LIN {X 0,Y 509.342,Z 622.742,A -85,B 0,C 180,E1 -5495.94,E2 -5495.94} C_VEL
LIN {X 0,Y 509.421,Z 617.168,A -85,B 0,C 180,E1 -5497.133,E2 -5497.133} C_VEL
LIN {X 0,Y 509.56,Z 611.515,A -85,B 0,C 180,E1 -5498.127,E2 -5498.127} C_VEL
LIN {X 0,Y 509.746,Z 604.71,A -85,B 0,C 180,E1 -5499.123,E2 -5499.123} C_VEL
LIN {X 0,Y 509.975,Z 596.49,A -85,B 0,C 180,E1 -5500.12,E2 -5500.12} C_VEL
LIN {X 0,Y 510.261,Z 588.661,A -85,B 0,C 180,E1 -5500.917,E2 -5500.917} C_VEL
LIN {X 0,Y 510.548,Z 580.574,A -85,B 0,C 180,E1 -5501.614,E2 -5501.614} C_VEL
LIN {X 0,Y 510.783,Z 570.465,A -85,B 0,C 180,E1 -5502.336,E2 -5502.336} C_VEL
LIN {X 0,Y 511.032,Z 562.413,A -85,B 0,C 180,E1 -5502.813,E2 -5502.813} C_VEL
LIN {X 0,Y 511.32,Z 551.902,A -85,B 0,C 180,E1 -5503.31,E2 -5503.31} C_VEL
LIN {X 0,Y 511.513,Z 541.564,A -85,B 0,C 180,E1 -5503.685,E2 -5503.685} C_VEL
LIN {X 0,Y 511.738,Z 530.84,A -85,B 0,C 180,E1 -5503.957,E2 -5503.957} C_VEL
LIN {X 0,Y 511.952,Z 508.063,A -85,B 0,C 180,E1 -5504.306,E2 -5504.306} C_VEL
LIN {X 0,Y 512.118,Z 435.713,A -85,B 0,C 180,E1 -5505.329,E2 -5505.329} C_VEL
LIN {X 0,Y 510.056,Z 423.426,A -85,B 0,C 180,E1 -5505.593,E2 -5505.593} C_VEL
LIN {X 0,Y 510.461,Z 407.833,A -85,B 0,C 180,E1 -5508.669,E2 -5508.669} C_VEL
LIN {X 0,Y 510.875,Z 391.094,A -85,B 0,C 180,E1 -5512.016,E2 -5512.016} C_VEL
LIN {X 0,Y 511.227,Z 378.573,A -85,B 0,C 180,E1 -5514.597,E2 -5514.597} C_VEL
LIN {X 0,Y 509.916,Z 370.577,A -85,B 0,C 180,E1 -5516.406,E2 -5516.406} C_VEL
LIN {X 0,Y 509.885,Z 370.471,A -85,B 0,C 180,E1 -5518.844,E2 -5518.844} C_VEL
LIN {X 0,Y 509.826,Z 370.48,A -85,B 0,C 180,E1 -5521.59,E2 -5521.59} C_VEL
LIN {X 0,Y 509.857,Z 370.474,A -85,B 0,C 180,E1 -5524.413,E2 -5524.413} C_VEL
LIN {X 0,Y 509.822,Z 370.475,A -85,B 0,C 180,E1 -5527.34,E2 -5527.34} C_VEL
LIN {X 0,Y 509.84,Z 370.468,A -85,B 0,C 180,E1 -5530.382,E2 -5530.382} C_VEL
LIN {X 0,Y 509.825,Z 370.474,A -85,B 0,C 180,E1 -5533.062,E2 -5533.062} C_VEL
LIN {X 0,Y 509.832,Z 370.478,A -85,B 0,C 180,E1 -5535.792,E2 -5535.792} C_VEL
LIN {X 0,Y 509.867,Z 370.469,A -85,B 0,C 180,E1 -5538.575,E2 -5538.575} C_VEL
LIN {X 0,Y 509.853,Z 370.475,A -85,B 0,C 180,E1 -5541.786,E2 -5541.786} C_VEL
LIN {X 0,Y 509.843,Z 370.47,A -85,B 0,C 180,E1 -5544.622,E2 -5544.622} C_VEL
LIN {X 0,Y 509.866,Z 370.468,A -85,B 0,C 180,E1 -5547.481,E2 -5547.481} C_VEL
LIN {X 0,Y 509.882,Z 370.469,A -85,B 0,C 180,E1 -5550.268,E2 -5550.268} C_VEL
LIN {X 0,Y 509.885,Z 370.459,A -85,B 0,C 180,E1 -5552.944,E2 -5552.944} C_VEL
LIN {X 0,Y 509.869,Z 370.47,A -85,B 0,C 180,E1 -5555.574,E2 -5555.574} C_VEL
LIN {X 0,Y 509.821,Z 370.477,A -85,B 0,C 180,E1 -5558.148,E2 -5558.148} C_VEL
LIN {X 0,Y 509.864,Z 370.461,A -85,B 0,C 180,E1 -5560.681,E2 -5560.681} C_VEL
LIN {X 0,Y 509.884,Z 370.462,A -85,B 0,C 180,E1 -5563.174,E2 -5563.174} C_VEL
LIN {X 0,Y 509.863,Z 370.475,A -85,B 0,C 180,E1 -5565.634,E2 -5565.634} C_VEL
LIN {X 0,Y 509.911,Z 370.458,A -85,B 0,C 180,E1 -5568.874,E2 -5568.874} C_VEL
LIN {X 0,Y 509.95,Z 370.458,A -85,B 0,C 180,E1 -5572.078,E2 -5572.078} C_VEL
LIN {X 0,Y 509.98,Z 370.455,A -85,B 0,C 180,E1 -5574.464,E2 -5574.464} C_VEL
LIN {X 0,Y 510.053,Z 370.45,A -85,B 0,C 180,E1 -5577.63,E2 -5577.63} C_VEL
LIN {X 0,Y 510.062,Z 370.433,A -85,B 0,C 180,E1 -5580.789,E2 -5580.789} C_VEL
LIN {X 0,Y 509.955,Z 370.457,A -85,B 0,C 180,E1 -5583.16,E2 -5583.16} C_VEL
LIN {X 0,Y 509.975,Z 370.455,A -85,B 0,C 180,E1 -5586.329,E2 -5586.329} C_VEL
LIN {X 0,Y 509.913,Z 370.457,A -85,B 0,C 180,E1 -5588.72,E2 -5588.72} C_VEL
LIN {X 0,Y 509.948,Z 370.46,A -85,B 0,C 180,E1 -5591.93,E2 -5591.93} C_VEL
LIN {X 0,Y 509.89,Z 370.471,A -85,B 0,C 180,E1 -5595.241,E2 -5595.241} C_VEL
LIN {X 0,Y 509.885,Z 370.461,A -85,B 0,C 180,E1 -5598.001,E2 -5598.001} C_VEL
LIN {X 0,Y 509.847,Z 370.468,A -85,B 0,C 180,E1 -5601.001,E2 -5601.001} C_VEL
LIN {X 0,Y 509.866,Z 370.469,A -85,B 0,C 180,E1 -5604.426,E2 -5604.426} C_VEL
LIN {X 0,Y 509.884,Z 370.465,A -85,B 0,C 180,E1 -5607.055,E2 -5607.055} C_VEL
LIN {X 0,Y 509.853,Z 370.475,A -85,B 0,C 180,E1 -5609.751,E2 -5609.751} C_VEL
LIN {X 0,Y 509.873,Z 370.469,A -85,B 0,C 180,E1 -5612.775,E2 -5612.775} C_VEL
LIN {X 0,Y 509.838,Z 370.478,A -85,B 0,C 180,E1 -5615.581,E2 -5615.581} C_VEL
LIN {X 0,Y 509.846,Z 370.472,A -85,B 0,C 180,E1 -5618.338,E2 -5618.338} C_VEL
LIN {X 0,Y 509.855,Z 370.475,A -85,B 0,C 180,E1 -5621.425,E2 -5621.425} C_VEL
LIN {X 0,Y 509.852,Z 370.471,A -85,B 0,C 180,E1 -5624.668,E2 -5624.668} C_VEL
LIN {X 0,Y 509.857,Z 370.456,A -85,B 0,C 180,E1 -5628.102,E2 -5628.102} C_VEL
LIN {X 0,Y 509.856,Z 370.469,A -85,B 0,C 180,E1 -5630.649,E2 -5630.649} C_VEL
LIN {X 0,Y 509.828,Z 370.472,A -85,B 0,C 180,E1 -5633.742,E2 -5633.742} C_VEL
LIN {X 0,Y 509.162,Z 370.553,A -85,B 0,C 180,E1 -5634.402,E2 -5634.402} C_VEL
LIN {X 0,Y 506.344,Z 370.904,A -85,B 0,C 180,E1 -5635.474,E2 -5635.474} C_VEL
LIN {X 0,Y 503.951,Z 371.205,A -85,B 0,C 180,E1 -5636.337,E2 -5636.337} C_VEL
LIN {X 0,Y 502.902,Z 371.337,A -85,B 0,C 180,E1 -5637.004,E2 -5637.004} C_VEL
LIN {X 0,Y 502.805,Z 371.348,A -85,B 0,C 180,E1 -5637.229,E2 -5637.229} C_VEL
LIN {X 0,Y 502.827,Z 371.341,A -85,B 0,C 180,E1 -5640.061,E2 -5640.061} C_VEL
LIN {X 0,Y 502.831,Z 371.347,A -85,B 0,C 180,E1 -5642.533,E2 -5642.533} C_VEL
LIN {X 0,Y 502.825,Z 371.354,A -85,B 0,C 180,E1 -5645.298,E2 -5645.298} C_VEL
LIN {X 0,Y 502.79,Z 371.354,A -85,B 0,C 180,E1 -5647.827,E2 -5647.827} C_VEL
LIN {X 0,Y 502.823,Z 371.349,A -85,B 0,C 180,E1 -5650.4,E2 -5650.4} C_VEL
LIN {X 0,Y 502.831,Z 371.353,A -85,B 0,C 180,E1 -5652.932,E2 -5652.932} C_VEL
LIN {X 0,Y 502.842,Z 371.351,A -85,B 0,C 180,E1 -5655.429,E2 -5655.429} C_VEL
LIN {X 0,Y 502.874,Z 371.347,A -85,B 0,C 180,E1 -5658.717,E2 -5658.717} C_VEL
LIN {X 0,Y 502.898,Z 371.34,A -85,B 0,C 180,E1 -5661.966,E2 -5661.966} C_VEL
LIN {X 0,Y 502.939,Z 371.336,A -85,B 0,C 180,E1 -5664.386,E2 -5664.386} C_VEL
LIN {X 0,Y 503.023,Z 371.326,A -85,B 0,C 180,E1 -5667.598,E2 -5667.598} C_VEL
LIN {X 0,Y 503.025,Z 371.324,A -85,B 0,C 180,E1 -5670,E2 -5670} C_VEL
LIN {X 0,Y 503.022,Z 371.326,A -85,B 0,C 180,E1 -5672.402,E2 -5672.402} C_VEL
LIN {X 0,Y 502.939,Z 371.336,A -85,B 0,C 180,E1 -5675.613,E2 -5675.613} C_VEL
LIN {X 0,Y 502.898,Z 371.34,A -85,B 0,C 180,E1 -5678.033,E2 -5678.033} C_VEL
LIN {X 0,Y 502.873,Z 371.347,A -85,B 0,C 180,E1 -5681.283,E2 -5681.283} C_VEL
LIN {X 0,Y 502.841,Z 371.351,A -85,B 0,C 180,E1 -5684.571,E2 -5684.571} C_VEL
LIN {X 0,Y 502.858,Z 371.344,A -85,B 0,C 180,E1 -5687.907,E2 -5687.907} C_VEL
LIN {X 0,Y 502.824,Z 371.353,A -85,B 0,C 180,E1 -5690.536,E2 -5690.536} C_VEL
LIN {X 0,Y 502.792,Z 371.358,A -85,B 0,C 180,E1 -5693.04,E2 -5693.04} C_VEL
LIN {X 0,Y 502.837,Z 371.347,A -85,B 0,C 180,E1 -5695.675,E2 -5695.675} C_VEL
LIN {X 0,Y 502.837,Z 371.349,A -85,B 0,C 180,E1 -5698.372,E2 -5698.372} C_VEL
LIN {X 0,Y 502.791,Z 371.352,A -85,B 0,C 180,E1 -5701.499,E2 -5701.499} C_VEL
LIN {X 0,Y 502.8,Z 371.346,A -85,B 0,C 180,E1 -5704.444,E2 -5704.444} C_VEL
LIN {X 0,Y 502.775,Z 371.356,A -85,B 0,C 180,E1 -5707.178,E2 -5707.178} C_VEL
LIN {X 0,Y 502.815,Z 371.346,A -85,B 0,C 180,E1 -5710.012,E2 -5710.012} C_VEL
LIN {X 0,Y 502.766,Z 371.348,A -85,B 0,C 180,E1 -5713.231,E2 -5713.231} C_VEL
LIN {X 0,Y 502.783,Z 371.351,A -85,B 0,C 180,E1 -5715.661,E2 -5715.661} C_VEL
LIN {X 0,Y 502.813,Z 371.348,A -85,B 0,C 180,E1 -5718.934,E2 -5718.934} C_VEL
LIN {X 0,Y 502.788,Z 371.353,A -85,B 0,C 180,E1 -5722.046,E2 -5722.046} C_VEL
LIN {X 0,Y 502.803,Z 371.345,A -85,B 0,C 180,E1 -5725.035,E2 -5725.035} C_VEL
LIN {X 0,Y 502.781,Z 371.352,A -85,B 0,C 180,E1 -5727.916,E2 -5727.916} C_VEL
LIN {X 0,Y 502.832,Z 371.347,A -85,B 0,C 180,E1 -5730.713,E2 -5730.713} C_VEL
LIN {X 0,Y 502.874,Z 371.335,A -85,B 0,C 180,E1 -5733.435,E2 -5733.435} C_VEL
LIN {X 0,Y 502.784,Z 371.354,A -85,B 0,C 180,E1 -5736.086,E2 -5736.086} C_VEL
LIN {X 0,Y 502.777,Z 371.353,A -85,B 0,C 180,E1 -5738.689,E2 -5738.689} C_VEL
LIN {X 0,Y 502.824,Z 371.338,A -85,B 0,C 180,E1 -5741.249,E2 -5741.249} C_VEL
LIN {X 0,Y 502.817,Z 371.346,A -85,B 0,C 180,E1 -5743.767,E2 -5743.767} C_VEL
LIN {X 0,Y 502.825,Z 371.352,A -85,B 0,C 180,E1 -5746.255,E2 -5746.255} C_VEL
LIN {X 0,Y 502.886,Z 371.333,A -85,B 0,C 180,E1 -5748.718,E2 -5748.718} C_VEL
LIN {X 0,Y 502.895,Z 371.334,A -85,B 0,C 180,E1 -5751.967,E2 -5751.967} C_VEL
LIN {X 0,Y 502.933,Z 371.341,A -85,B 0,C 180,E1 -5754.387,E2 -5754.387} C_VEL
LIN {X 0,Y 503.02,Z 371.318,A -85,B 0,C 180,E1 -5757.598,E2 -5757.598} C_VEL
LIN {X 0,Y 503.021,Z 371.313,A -85,B 0,C 180,E1 -5760,E2 -5760} C_VEL
LIN {X 0,Y 503.02,Z 371.327,A -85,B 0,C 180,E1 -5762.403,E2 -5762.403} C_VEL
LIN {X 0,Y 502.934,Z 371.333,A -85,B 0,C 180,E1 -5765.614,E2 -5765.614} C_VEL
LIN {X 0,Y 502.896,Z 371.338,A -85,B 0,C 180,E1 -5768.034,E2 -5768.034} C_VEL
LIN {X 0,Y 502.872,Z 371.335,A -85,B 0,C 180,E1 -5771.284,E2 -5771.284} C_VEL
LIN {X 0,Y 502.84,Z 371.347,A -85,B 0,C 180,E1 -5774.571,E2 -5774.571} C_VEL
LIN {X 0,Y 502.857,Z 371.339,A -85,B 0,C 180,E1 -5777.908,E2 -5777.908} C_VEL
LIN {X 0,Y 502.824,Z 371.348,A -85,B 0,C 180,E1 -5780.537,E2 -5780.537} C_VEL
LIN {X 0,Y 502.792,Z 371.35,A -85,B 0,C 180,E1 -5783.041,E2 -5783.041} C_VEL
LIN {X 0,Y 502.838,Z 371.343,A -85,B 0,C 180,E1 -5785.676,E2 -5785.676} C_VEL
LIN {X 0,Y 502.839,Z 371.349,A -85,B 0,C 180,E1 -5788.373,E2 -5788.373} C_VEL
LIN {X 0,Y 502.794,Z 371.351,A -85,B 0,C 180,E1 -5791.5,E2 -5791.5} C_VEL
LIN {X 0,Y 502.804,Z 371.35,A -85,B 0,C 180,E1 -5794.446,E2 -5794.446} C_VEL
LIN {X 0,Y 502.779,Z 371.352,A -85,B 0,C 180,E1 -5797.179,E2 -5797.179} C_VEL
LIN {X 0,Y 502.82,Z 371.35,A -85,B 0,C 180,E1 -5800.013,E2 -5800.013} C_VEL
LIN {X 0,Y 502.821,Z 371.353,A -85,B 0,C 180,E1 -5802.203,E2 -5802.203} C_VEL
LIN {X 0,Y 502.799,Z 371.351,A -85,B 0,C 180,E1 -5805.469,E2 -5805.469} C_VEL
LIN {X 0,Y 502.82,Z 371.339,A -85,B 0,C 180,E1 -5808.935,E2 -5808.935} C_VEL
LIN {X 0,Y 502.794,Z 371.358,A -85,B 0,C 180,E1 -5812.047,E2 -5812.047} C_VEL
LIN {X 0,Y 502.81,Z 371.348,A -85,B 0,C 180,E1 -5815.036,E2 -5815.036} C_VEL
LIN {X 0,Y 502.786,Z 371.356,A -85,B 0,C 180,E1 -5817.916,E2 -5817.916} C_VEL
LIN {X 0,Y 502.841,Z 371.349,A -85,B 0,C 180,E1 -5820.714,E2 -5820.714} C_VEL
LIN {X 0,Y 502.867,Z 371.475,A -85,B 0,C 180,E1 -5823.439,E2 -5823.439} C_VEL
LIN {X 0,Y 504.25,Z 379.576,A -85,B 0,C 180,E1 -5825.284,E2 -5825.284} C_VEL
LIN {X 0,Y 503.892,Z 393.054,A -85,B 0,C 180,E1 -5828.094,E2 -5828.094} C_VEL
LIN {X 0,Y 503.435,Z 408.697,A -85,B 0,C 180,E1 -5831.272,E2 -5831.272} C_VEL
LIN {X 0,Y 503.026,Z 423.045,A -85,B 0,C 180,E1 -5834.167,E2 -5834.167} C_VEL
LIN {X 0,Y 503.739,Z 427.556,A -85,B 0,C 180,E1 -5834.295,E2 -5834.295} C_VEL
LIN {X 0,Y 505.36,Z 437.202,A -85,B 0,C 180,E1 -5834.486,E2 -5834.486} C_VEL
LIN {X 0,Y 504.882,Z 528.027,A -85,B 0,C 180,E1 -5835.798,E2 -5835.798} C_VEL
LIN {X 0,Y 504.693,Z 537.941,A -85,B 0,C 180,E1 -5836.024,E2 -5836.024} C_VEL
LIN {X 0,Y 504.506,Z 547.93,A -85,B 0,C 180,E1 -5836.353,E2 -5836.353} C_VEL
LIN {X 0,Y 504.175,Z 558.287,A -85,B 0,C 180,E1 -5836.806,E2 -5836.806} C_VEL
LIN {X 0,Y 503.896,Z 568.156,A -85,B 0,C 180,E1 -5837.357,E2 -5837.357} C_VEL
LIN {X 0,Y 503.666,Z 576.443,A -85,B 0,C 180,E1 -5837.919,E2 -5837.919} C_VEL
LIN {X 0,Y 503.36,Z 585.173,A -85,B 0,C 180,E1 -5838.626,E2 -5838.626} C_VEL
LIN {X 0,Y 503.091,Z 592.597,A -85,B 0,C 180,E1 -5839.334,E2 -5839.334} C_VEL
LIN {X 0,Y 502.801,Z 601.396,A -85,B 0,C 180,E1 -5840.344,E2 -5840.344} C_VEL
LIN {X 0,Y 502.602,Z 607.387,A -85,B 0,C 180,E1 -5841.152,E2 -5841.152} C_VEL
LIN {X 0,Y 502.413,Z 613.697,A -85,B 0,C 180,E1 -5842.161,E2 -5842.161} C_VEL
LIN {X 0,Y 502.284,Z 619.149,A -85,B 0,C 180,E1 -5843.21,E2 -5843.21} C_VEL
LIN {X 0,Y 502.217,Z 624.061,A -85,B 0,C 180,E1 -5844.379,E2 -5844.379} C_VEL
LIN {X 0,Y 502.103,Z 628.019,A -85,B 0,C 180,E1 -5845.585,E2 -5845.585} C_VEL
LIN {X 0,Y 502.12,Z 630.949,A -85,B 0,C 180,E1 -5846.791,E2 -5846.791} C_VEL
LIN {X 0,Y 502.091,Z 632.445,A -85,B 0,C 180,E1 -5847.594,E2 -5847.594} C_VEL
LIN {X 0,Y 501.99,Z 633.96,A -85,B 0,C 180,E1 -5849.198,E2 -5849.198} C_VEL
LIN {X 0,Y 501.98,Z 634.238,A -85,B 0,C 180,E1 -5850,E2 -5850} C_VEL
LIN {X 0,Y 502.036,Z 633.367,A -85,B 0,C 180,E1 -5851.605,E2 -5851.605} C_VEL
LIN {X 0,Y 502.091,Z 632.444,A -85,B 0,C 180,E1 -5852.407,E2 -5852.407} C_VEL
LIN {X 0,Y 502.139,Z 629.106,A -85,B 0,C 180,E1 -5854.013,E2 -5854.013} C_VEL
LIN {X 0,Y 502.175,Z 625.485,A -85,B 0,C 180,E1 -5855.219,E2 -5855.219} C_VEL
LIN {X 0,Y 502.236,Z 620.757,A -85,B 0,C 180,E1 -5856.428,E2 -5856.428} C_VEL
LIN {X 0,Y 502.36,Z 615.88,A -85,B 0,C 180,E1 -5857.435,E2 -5857.435} C_VEL
LIN {X 0,Y 502.516,Z 610.007,A -85,B 0,C 180,E1 -5858.445,E2 -5858.445} C_VEL
LIN {X 0,Y 502.683,Z 604.514,A -85,B 0,C 180,E1 -5859.252,E2 -5859.252} C_VEL
LIN {X 0,Y 502.945,Z 596.294,A -85,B 0,C 180,E1 -5860.263,E2 -5860.263} C_VEL
LIN {X 0,Y 503.253,Z 588.465,A -85,B 0,C 180,E1 -5861.071,E2 -5861.071} C_VEL
LIN {X 0,Y 503.575,Z 580.379,A -85,B 0,C 180,E1 -5861.777,E2 -5861.777} C_VEL
LIN {X 0,Y 503.79,Z 571.355,A -85,B 0,C 180,E1 -5862.44,E2 -5862.44} C_VEL
LIN {X 0,Y 504.082,Z 562.217,A -85,B 0,C 180,E1 -5862.992,E2 -5862.992} C_VEL
LIN {X 0,Y 504.396,Z 551.706,A -85,B 0,C 180,E1 -5863.497,E2 -5863.497} C_VEL
LIN {X 0,Y 504.627,Z 541.369,A -85,B 0,C 180,E1 -5863.875,E2 -5863.875} C_VEL
LIN {X 0,Y 504.87,Z 530.646,A -85,B 0,C 180,E1 -5864.151,E2 -5864.151} C_VEL
LIN {X 0,Y 505.055,Z 507.867,A -85,B 0,C 180,E1 -5864.506,E2 -5864.506} C_VEL
LIN {X 0,Y 505.304,Z 436.726,A -85,B 0,C 180,E1 -5865.523,E2 -5865.523} C_VEL
LIN {X 0,Y 503.049,Z 423.383,A -85,B 0,C 180,E1 -5865.805,E2 -5865.805} C_VEL
LIN {X 0,Y 503.028,Z 422.359,A -85,B 0,C 180,E1 -5865.945,E2 -5865.945} C_VEL
LIN {X 0,Y 503.457,Z 407.697,A -85,B 0,C 180,E1 -5868.939,E2 -5868.939} C_VEL
LIN {X 0,Y 503.889,Z 392.003,A -85,B 0,C 180,E1 -5872.122,E2 -5872.122} C_VEL
LIN {X 0,Y 504.274,Z 379.608,A -85,B 0,C 180,E1 -5874.715,E2 -5874.715} C_VEL
LIN {X 0,Y 502.885,Z 371.469,A -85,B 0,C 180,E1 -5876.565,E2 -5876.565} C_VEL
LIN {X 0,Y 502.84,Z 371.349,A -85,B 0,C 180,E1 -5879.287,E2 -5879.287} C_VEL
LIN {X 0,Y 502.788,Z 371.356,A -85,B 0,C 180,E1 -5882.084,E2 -5882.084} C_VEL
LIN {X 0,Y 502.812,Z 371.348,A -85,B 0,C 180,E1 -5884.965,E2 -5884.965} C_VEL
LIN {X 0,Y 502.796,Z 371.357,A -85,B 0,C 180,E1 -5887.953,E2 -5887.953} C_VEL
LIN {X 0,Y 502.822,Z 371.338,A -85,B 0,C 180,E1 -5891.065,E2 -5891.065} C_VEL
LIN {X 0,Y 502.802,Z 371.35,A -85,B 0,C 180,E1 -5894.531,E2 -5894.531} C_VEL
LIN {X 0,Y 502.836,Z 371.352,A -85,B 0,C 180,E1 -5897.864,E2 -5897.864} C_VEL
LIN {X 0,Y 502.81,Z 371.345,A -85,B 0,C 180,E1 -5901.024,E2 -5901.024} C_VEL
LIN {X 0,Y 502.783,Z 371.353,A -85,B 0,C 180,E1 -5904.167,E2 -5904.167} C_VEL
LIN {X 0,Y 502.833,Z 371.341,A -85,B 0,C 180,E1 -5906.993,E2 -5906.993} C_VEL
LIN {X 0,Y 502.831,Z 371.35,A -85,B 0,C 180,E1 -5910.061,E2 -5910.061} C_VEL
LIN {X 0,Y 502.834,Z 371.338,A -85,B 0,C 180,E1 -5912.533,E2 -5912.533} C_VEL
LIN {X 0,Y 502.828,Z 371.344,A -85,B 0,C 180,E1 -5915.298,E2 -5915.298} C_VEL
LIN {X 0,Y 502.784,Z 371.358,A -85,B 0,C 180,E1 -5917.826,E2 -5917.826} C_VEL
LIN {X 0,Y 502.824,Z 371.339,A -85,B 0,C 180,E1 -5920.4,E2 -5920.4} C_VEL
LIN {X 0,Y 502.833,Z 371.338,A -85,B 0,C 180,E1 -5922.931,E2 -5922.931} C_VEL
LIN {X 0,Y 502.844,Z 371.346,A -85,B 0,C 180,E1 -5925.429,E2 -5925.429} C_VEL
LIN {X 0,Y 502.875,Z 371.334,A -85,B 0,C 180,E1 -5928.716,E2 -5928.716} C_VEL
LIN {X 0,Y 502.9,Z 371.337,A -85,B 0,C 180,E1 -5931.966,E2 -5931.966} C_VEL
LIN {X 0,Y 502.936,Z 371.333,A -85,B 0,C 180,E1 -5934.386,E2 -5934.386} C_VEL
LIN {X 0,Y 503.022,Z 371.326,A -85,B 0,C 180,E1 -5937.597,E2 -5937.597} C_VEL
LIN {X 0,Y 503.025,Z 371.313,A -85,B 0,C 180,E1 -5940,E2 -5940} C_VEL
LIN {X 0,Y 503.022,Z 371.318,A -85,B 0,C 180,E1 -5942.402,E2 -5942.402} C_VEL
LIN {X 0,Y 502.936,Z 371.341,A -85,B 0,C 180,E1 -5945.613,E2 -5945.613} C_VEL
LIN {X 0,Y 502.899,Z 371.333,A -85,B 0,C 180,E1 -5948.033,E2 -5948.033} C_VEL
LIN {X 0,Y 502.889,Z 371.332,A -85,B 0,C 180,E1 -5951.282,E2 -5951.282} C_VEL
LIN {X 0,Y 502.842,Z 371.344,A -85,B 0,C 180,E1 -5954.57,E2 -5954.57} C_VEL
LIN {X 0,Y 502.858,Z 371.337,A -85,B 0,C 180,E1 -5957.907,E2 -5957.907} C_VEL
LIN {X 0,Y 502.825,Z 371.34,A -85,B 0,C 180,E1 -5960.536,E2 -5960.536} C_VEL
LIN {X 0,Y 502.79,Z 371.353,A -85,B 0,C 180,E1 -5963.04,E2 -5963.04} C_VEL
LIN {X 0,Y 502.838,Z 371.345,A -85,B 0,C 180,E1 -5965.675,E2 -5965.675} C_VEL
LIN {X 0,Y 502.837,Z 371.34,A -85,B 0,C 180,E1 -5968.372,E2 -5968.372} C_VEL
LIN {X 0,Y 502.792,Z 371.358,A -85,B 0,C 180,E1 -5971.499,E2 -5971.499} C_VEL
LIN {X 0,Y 502.802,Z 371.342,A -85,B 0,C 180,E1 -5974.444,E2 -5974.444} C_VEL
LIN {X 0,Y 502.777,Z 371.357,A -85,B 0,C 180,E1 -5977.178,E2 -5977.178} C_VEL
LIN {X 0,Y 502.784,Z 371.348,A -85,B 0,C 180,E1 -5980.015,E2 -5980.015} C_VEL
LIN {X 0,Y 502.799,Z 371.349,A -85,B 0,C 180,E1 -5982.199,E2 -5982.199} C_VEL
LIN {X 0,Y 502.796,Z 371.349,A -85,B 0,C 180,E1 -5985.468,E2 -5985.468} C_VEL
LIN {X 0,Y 502.822,Z 371.336,A -85,B 0,C 180,E1 -5989.004,E2 -5989.004} C_VEL
LIN {X 0,Y 502.791,Z 371.352,A -85,B 0,C 180,E1 -5992.046,E2 -5992.046} C_VEL
LIN {X 0,Y 502.806,Z 371.346,A -85,B 0,C 180,E1 -5995.035,E2 -5995.035} C_VEL
LIN {X 0,Y 502.805,Z 371.348,A -85,B 0,C 180,E1 -5997.229,E2 -5997.229} C_VEL
LIN {X 0,Y 502.108,Z 371.439,A -85,B 0,C 180,E1 -5997.898,E2 -5997.898} C_VEL
LIN {X 0,Y 499.25,Z 371.798,A -85,B 0,C 180,E1 -5998.984,E2 -5998.984} C_VEL
LIN {X 0,Y 496.858,Z 372.089,A -85,B 0,C 180,E1 -5999.859,E2 -5999.859} C_VEL
LIN {X 0,Y 495.841,Z 372.212,A -85,B 0,C 180,E1 -6000.535,E2 -6000.535} C_VEL
LIN {X 0,Y 495.761,Z 372.221,A -85,B 0,C 180,E1 -6000.763,E2 -6000.763} C_VEL
LIN {X 0,Y 495.787,Z 372.225,A -85,B 0,C 180,E1 -6003.932,E2 -6003.932} C_VEL
LIN {X 0,Y 495.755,Z 372.235,A -85,B 0,C 180,E1 -6007.139,E2 -6007.139} C_VEL
LIN {X 0,Y 495.775,Z 372.227,A -85,B 0,C 180,E1 -6010.11,E2 -6010.11} C_VEL
LIN {X 0,Y 495.784,Z 372.229,A -85,B 0,C 180,E1 -6012.681,E2 -6012.681} C_VEL
LIN {X 0,Y 495.787,Z 372.231,A -85,B 0,C 180,E1 -6015.217,E2 -6015.217} C_VEL
LIN {X 0,Y 495.848,Z 372.22,A -85,B 0,C 180,E1 -6018.555,E2 -6018.555} C_VEL
LIN {X 0,Y 495.87,Z 372.216,A -85,B 0,C 180,E1 -6021.852,E2 -6021.852} C_VEL
LIN {X 0,Y 495.896,Z 372.213,A -85,B 0,C 180,E1 -6024.306,E2 -6024.306} C_VEL
LIN {X 0,Y 495.991,Z 372.202,A -85,B 0,C 180,E1 -6027.563,E2 -6027.563} C_VEL
LIN {X 0,Y 495.996,Z 372.2,A -85,B 0,C 180,E1 -6030,E2 -6030} C_VEL
LIN {X 0,Y 495.991,Z 372.202,A -85,B 0,C 180,E1 -6032.436,E2 -6032.436} C_VEL
LIN {X 0,Y 495.896,Z 372.213,A -85,B 0,C 180,E1 -6035.693,E2 -6035.693} C_VEL
LIN {X 0,Y 495.869,Z 372.216,A -85,B 0,C 180,E1 -6038.148,E2 -6038.148} C_VEL
LIN {X 0,Y 495.848,Z 372.22,A -85,B 0,C 180,E1 -6041.445,E2 -6041.445} C_VEL
LIN {X 0,Y 495.786,Z 372.231,A -85,B 0,C 180,E1 -6044.783,E2 -6044.783} C_VEL
LIN {X 0,Y 495.783,Z 372.229,A -85,B 0,C 180,E1 -6047.318,E2 -6047.318} C_VEL
LIN {X 0,Y 495.774,Z 372.227,A -85,B 0,C 180,E1 -6049.89,E2 -6049.89} C_VEL
LIN {X 0,Y 495.753,Z 372.236,A -85,B 0,C 180,E1 -6052.86,E2 -6052.86} C_VEL
LIN {X 0,Y 495.794,Z 372.224,A -85,B 0,C 180,E1 -6056.067,E2 -6056.067} C_VEL
LIN {X 0,Y 495.775,Z 372.224,A -85,B 0,C 180,E1 -6058.814,E2 -6058.814} C_VEL
LIN {X 0,Y 495.753,Z 372.229,A -85,B 0,C 180,E1 -6061.726,E2 -6061.726} C_VEL
LIN {X 0,Y 495.77,Z 372.22,A -85,B 0,C 180,E1 -6064.695,E2 -6064.695} C_VEL
LIN {X 0,Y 495.725,Z 372.232,A -85,B 0,C 180,E1 -6067.561,E2 -6067.561} C_VEL
LIN {X 0,Y 495.773,Z 372.217,A -85,B 0,C 180,E1 -6070.698,E2 -6070.698} C_VEL
LIN {X 0,Y 495.727,Z 372.223,A -85,B 0,C 180,E1 -6074.001,E2 -6074.001} C_VEL
LIN {X 0,Y 495.727,Z 372.233,A -85,B 0,C 180,E1 -6077.118,E2 -6077.118} C_VEL
LIN {X 0,Y 495.752,Z 372.223,A -85,B 0,C 180,E1 -6079.953,E2 -6079.953} C_VEL
LIN {X 0,Y 495.726,Z 372.239,A -85,B 0,C 180,E1 -6082.552,E2 -6082.552} C_VEL
LIN {X 0,Y 495.778,Z 372.217,A -85,B 0,C 180,E1 -6085.457,E2 -6085.457} C_VEL
LIN {X 0,Y 495.753,Z 372.232,A -85,B 0,C 180,E1 -6088.364,E2 -6088.364} C_VEL
LIN {X 0,Y 495.783,Z 372.218,A -85,B 0,C 180,E1 -6091.506,E2 -6091.506} C_VEL
LIN {X 0,Y 495.792,Z 372.218,A -85,B 0,C 180,E1 -6093.933,E2 -6093.933} C_VEL
LIN {X 0,Y 495.758,Z 372.227,A -85,B 0,C 180,E1 -6097.138,E2 -6097.138} C_VEL
LIN {X 0,Y 495.771,Z 372.222,A -85,B 0,C 180,E1 -6100.11,E2 -6100.11} C_VEL
LIN {X 0,Y 495.782,Z 372.228,A -85,B 0,C 180,E1 -6102.682,E2 -6102.682} C_VEL
LIN {X 0,Y 495.783,Z 372.224,A -85,B 0,C 180,E1 -6105.217,E2 -6105.217} C_VEL
LIN {X 0,Y 495.861,Z 372.209,A -85,B 0,C 180,E1 -6108.556,E2 -6108.556} C_VEL
LIN {X 0,Y 495.866,Z 372.208,A -85,B 0,C 180,E1 -6111.852,E2 -6111.852} C_VEL
LIN {X 0,Y 495.89,Z 372.217,A -85,B 0,C 180,E1 -6114.307,E2 -6114.307} C_VEL
LIN {X 0,Y 495.988,Z 372.194,A -85,B 0,C 180,E1 -6117.564,E2 -6117.564} C_VEL
LIN {X 0,Y 495.992,Z 372.188,A -85,B 0,C 180,E1 -6120,E2 -6120} C_VEL
LIN {X 0,Y 495.988,Z 372.203,A -85,B 0,C 180,E1 -6122.437,E2 -6122.437} C_VEL
LIN {X 0,Y 495.891,Z 372.211,A -85,B 0,C 180,E1 -6125.694,E2 -6125.694} C_VEL
LIN {X 0,Y 495.867,Z 372.211,A -85,B 0,C 180,E1 -6128.148,E2 -6128.148} C_VEL
LIN {X 0,Y 495.846,Z 372.21,A -85,B 0,C 180,E1 -6131.446,E2 -6131.446} C_VEL
LIN {X 0,Y 495.785,Z 372.223,A -85,B 0,C 180,E1 -6134.783,E2 -6134.783} C_VEL
LIN {X 0,Y 495.783,Z 372.216,A -85,B 0,C 180,E1 -6137.319,E2 -6137.319} C_VEL
LIN {X 0,Y 495.773,Z 372.219,A -85,B 0,C 180,E1 -6139.891,E2 -6139.891} C_VEL
LIN {X 0,Y 495.761,Z 372.226,A -85,B 0,C 180,E1 -6142.863,E2 -6142.863} C_VEL
LIN {X 0,Y 495.796,Z 372.22,A -85,B 0,C 180,E1 -6146.068,E2 -6146.068} C_VEL
LIN {X 0,Y 495.777,Z 372.224,A -85,B 0,C 180,E1 -6148.815,E2 -6148.815} C_VEL
LIN {X 0,Y 495.756,Z 372.23,A -85,B 0,C 180,E1 -6151.727,E2 -6151.727} C_VEL
LIN {X 0,Y 495.774,Z 372.223,A -85,B 0,C 180,E1 -6154.696,E2 -6154.696} C_VEL
LIN {X 0,Y 495.729,Z 372.233,A -85,B 0,C 180,E1 -6157.562,E2 -6157.562} C_VEL
LIN {X 0,Y 495.778,Z 372.224,A -85,B 0,C 180,E1 -6160.699,E2 -6160.699} C_VEL
LIN {X 0,Y 495.733,Z 372.234,A -85,B 0,C 180,E1 -6163.696,E2 -6163.696} C_VEL
LIN {X 0,Y 495.727,Z 372.235,A -85,B 0,C 180,E1 -6166.306,E2 -6166.306} C_VEL
LIN {X 0,Y 495.766,Z 372.218,A -85,B 0,C 180,E1 -6169.301,E2 -6169.301} C_VEL
LIN {X 0,Y 495.731,Z 372.232,A -85,B 0,C 180,E1 -6172.439,E2 -6172.439} C_VEL
LIN {X 0,Y 495.786,Z 372.225,A -85,B 0,C 180,E1 -6175.458,E2 -6175.458} C_VEL
LIN {X 0,Y 495.758,Z 372.233,A -85,B 0,C 180,E1 -6178.365,E2 -6178.365} C_VEL
LIN {X 0,Y 495.792,Z 372.228,A -85,B 0,C 180,E1 -6181.507,E2 -6181.507} C_VEL
LIN {X 0,Y 495.829,Z 372.355,A -85,B 0,C 180,E1 -6183.25,E2 -6183.25} C_VEL
LIN {X 0,Y 497.25,Z 380.496,A -85,B 0,C 180,E1 -6185.136,E2 -6185.136} C_VEL
LIN {X 0,Y 497.036,Z 390.005,A -85,B 0,C 180,E1 -6187.166,E2 -6187.166} C_VEL
LIN {X 0,Y 496.554,Z 404.393,A -85,B 0,C 180,E1 -6190.143,E2 -6190.143} C_VEL
LIN {X 0,Y 496.12,Z 418.849,A -85,B 0,C 180,E1 -6193.118,E2 -6193.118} C_VEL
LIN {X 0,Y 496.005,Z 422.88,A -85,B 0,C 180,E1 -6193.94,E2 -6193.94} C_VEL
LIN {X 0,Y 496.799,Z 427.969,A -85,B 0,C 180,E1 -6194.079,E2 -6194.079} C_VEL
LIN {X 0,Y 498.546,Z 438.598,A -85,B 0,C 180,E1 -6194.291,E2 -6194.291} C_VEL
LIN {X 0,Y 498.009,Z 527.832,A -85,B 0,C 180,E1 -6195.598,E2 -6195.598} C_VEL
LIN {X 0,Y 497.815,Z 537.746,A -85,B 0,C 180,E1 -6195.827,E2 -6195.827} C_VEL
LIN {X 0,Y 497.609,Z 547.735,A -85,B 0,C 180,E1 -6196.16,E2 -6196.16} C_VEL
LIN {X 0,Y 497.254,Z 558.092,A -85,B 0,C 180,E1 -6196.619,E2 -6196.619} C_VEL
LIN {X 0,Y 496.996,Z 566.928,A -85,B 0,C 180,E1 -6197.111,E2 -6197.111} C_VEL
LIN {X 0,Y 496.685,Z 576.247,A -85,B 0,C 180,E1 -6197.746,E2 -6197.746} C_VEL
LIN {X 0,Y 496.386,Z 584.978,A -85,B 0,C 180,E1 -6198.464,E2 -6198.464} C_VEL
LIN {X 0,Y 496.104,Z 592.402,A -85,B 0,C 180,E1 -6199.182,E2 -6199.182} C_VEL
LIN {X 0,Y 495.754,Z 601.199,A -85,B 0,C 180,E1 -6200.206,E2 -6200.206} C_VEL
LIN {X 0,Y 495.565,Z 607.191,A -85,B 0,C 180,E1 -6201.026,E2 -6201.026} C_VEL
LIN {X 0,Y 495.363,Z 613.502,A -85,B 0,C 180,E1 -6202.049,E2 -6202.049} C_VEL
LIN {X 0,Y 495.223,Z 618.774,A -85,B 0,C 180,E1 -6203.072,E2 -6203.072} C_VEL
LIN {X 0,Y 495.136,Z 623.866,A -85,B 0,C 180,E1 -6204.298,E2 -6204.298} C_VEL
LIN {X 0,Y 495.009,Z 627.823,A -85,B 0,C 180,E1 -6205.522,E2 -6205.522} C_VEL
LIN {X 0,Y 495.042,Z 630.754,A -85,B 0,C 180,E1 -6206.745,E2 -6206.745} C_VEL
LIN {X 0,Y 494.998,Z 632.25,A -85,B 0,C 180,E1 -6207.559,E2 -6207.559} C_VEL
LIN {X 0,Y 494.911,Z 633.765,A -85,B 0,C 180,E1 -6209.187,E2 -6209.187} C_VEL
LIN {X 0,Y 494.898,Z 634.043,A -85,B 0,C 180,E1 -6210,E2 -6210} C_VEL
LIN {X 0,Y 494.963,Z 633.173,A -85,B 0,C 180,E1 -6211.628,E2 -6211.628} C_VEL
LIN {X 0,Y 494.998,Z 632.249,A -85,B 0,C 180,E1 -6212.441,E2 -6212.441} C_VEL
LIN {X 0,Y 495.032,Z 628.91,A -85,B 0,C 180,E1 -6214.071,E2 -6214.071} C_VEL
LIN {X 0,Y 495.108,Z 625.29,A -85,B 0,C 180,E1 -6215.294,E2 -6215.294} C_VEL
LIN {X 0,Y 495.136,Z 621.737,A -85,B 0,C 180,E1 -6216.251,E2 -6216.251} C_VEL
LIN {X 0,Y 495.307,Z 615.684,A -85,B 0,C 180,E1 -6217.542,E2 -6217.542} C_VEL
LIN {X 0,Y 495.474,Z 609.812,A -85,B 0,C 180,E1 -6218.565,E2 -6218.565} C_VEL
LIN {X 0,Y 495.628,Z 604.317,A -85,B 0,C 180,E1 -6219.385,E2 -6219.385} C_VEL
LIN {X 0,Y 495.928,Z 596.098,A -85,B 0,C 180,E1 -6220.41,E2 -6220.41} C_VEL
LIN {X 0,Y 496.265,Z 588.269,A -85,B 0,C 180,E1 -6221.229,E2 -6221.229} C_VEL
LIN {X 0,Y 496.602,Z 580.183,A -85,B 0,C 180,E1 -6221.945,E2 -6221.945} C_VEL
LIN {X 0,Y 496.82,Z 572.067,A -85,B 0,C 180,E1 -6222.558,E2 -6222.558} C_VEL
LIN {X 0,Y 497.161,Z 562.021,A -85,B 0,C 180,E1 -6223.176,E2 -6223.176} C_VEL
LIN {X 0,Y 497.501,Z 551.511,A -85,B 0,C 180,E1 -6223.687,E2 -6223.687} C_VEL
LIN {X 0,Y 497.712,Z 541.173,A -85,B 0,C 180,E1 -6224.072,E2 -6224.072} C_VEL
LIN {X 0,Y 497.997,Z 530.451,A -85,B 0,C 180,E1 -6224.35,E2 -6224.35} C_VEL
LIN {X 0,Y 498.181,Z 507.672,A -85,B 0,C 180,E1 -6224.71,E2 -6224.71} C_VEL
LIN {X 0,Y 498.478,Z 437.639,A -85,B 0,C 180,E1 -6225.725,E2 -6225.725} C_VEL
LIN {X 0,Y 496.044,Z 423.225,A -85,B 0,C 180,E1 -6226.033,E2 -6226.033} C_VEL
LIN {X 0,Y 496.041,Z 421.831,A -85,B 0,C 180,E1 -6226.25,E2 -6226.25} C_VEL
LIN {X 0,Y 496.442,Z 407.561,A -85,B 0,C 180,E1 -6229.217,E2 -6229.217} C_VEL
LIN {X 0,Y 496.929,Z 392.914,A -85,B 0,C 180,E1 -6232.23,E2 -6232.23} C_VEL
LIN {X 0,Y 497.34,Z 381.56,A -85,B 0,C 180,E1 -6234.637,E2 -6234.637} C_VEL
LIN {X 0,Y 496.381,Z 375.364,A -85,B 0,C 180,E1 -6236.034,E2 -6236.034} C_VEL
LIN {X 0,Y 495.824,Z 372.352,A -85,B 0,C 180,E1 -6236.748,E2 -6236.748} C_VEL
LIN {X 0,Y 495.784,Z 372.228,A -85,B 0,C 180,E1 -6239.745,E2 -6239.745} C_VEL
LIN {X 0,Y 495.796,Z 372.222,A -85,B 0,C 180,E1 -6243.244,E2 -6243.244} C_VEL
LIN {X 0,Y 495.731,Z 372.231,A -85,B 0,C 180,E1 -6246.09,E2 -6246.09} C_VEL
LIN {X 0,Y 495.766,Z 372.226,A -85,B 0,C 180,E1 -6248.768,E2 -6248.768} C_VEL
LIN {X 0,Y 495.76,Z 372.223,A -85,B 0,C 180,E1 -6251.78,E2 -6251.78} C_VEL
LIN {X 0,Y 495.751,Z 372.227,A -85,B 0,C 180,E1 -6255.139,E2 -6255.139} C_VEL
LIN {X 0,Y 495.783,Z 372.227,A -85,B 0,C 180,E1 -6258.221,E2 -6258.221} C_VEL
LIN {X 0,Y 495.769,Z 372.223,A -85,B 0,C 180,E1 -6261.23,E2 -6261.23} C_VEL
LIN {X 0,Y 495.755,Z 372.225,A -85,B 0,C 180,E1 -6264.462,E2 -6264.462} C_VEL
LIN {X 0,Y 495.77,Z 372.223,A -85,B 0,C 180,E1 -6267.405,E2 -6267.405} C_VEL
LIN {X 0,Y 495.782,Z 372.226,A -85,B 0,C 180,E1 -6270.254,E2 -6270.254} C_VEL
LIN {X 0,Y 495.823,Z 372.211,A -85,B 0,C 180,E1 -6273.25,E2 -6273.25} C_VEL
LIN {X 0,Y 495.752,Z 372.23,A -85,B 0,C 180,E1 -6275.725,E2 -6275.725} C_VEL
LIN {X 0,Y 495.743,Z 372.228,A -85,B 0,C 180,E1 -6278.371,E2 -6278.371} C_VEL
LIN {X 0,Y 495.784,Z 372.214,A -85,B 0,C 180,E1 -6280.971,E2 -6280.971} C_VEL
LIN {X 0,Y 495.778,Z 372.222,A -85,B 0,C 180,E1 -6283.53,E2 -6283.53} C_VEL
LIN {X 0,Y 495.792,Z 372.225,A -85,B 0,C 180,E1 -6286.055,E2 -6286.055} C_VEL
LIN {X 0,Y 495.85,Z 372.209,A -85,B 0,C 180,E1 -6288.554,E2 -6288.554} C_VEL
LIN {X 0,Y 495.871,Z 372.21,A -85,B 0,C 180,E1 -6291.852,E2 -6291.852} C_VEL
LIN {X 0,Y 495.894,Z 372.211,A -85,B 0,C 180,E1 -6294.306,E2 -6294.306} C_VEL
LIN {X 0,Y 495.991,Z 372.202,A -85,B 0,C 180,E1 -6297.563,E2 -6297.563} C_VEL
LIN {X 0,Y 495.996,Z 372.187,A -85,B 0,C 180,E1 -6300,E2 -6300} C_VEL
LIN {X 0,Y 495.991,Z 372.193,A -85,B 0,C 180,E1 -6302.436,E2 -6302.436} C_VEL
LIN {X 0,Y 495.893,Z 372.216,A -85,B 0,C 180,E1 -6305.693,E2 -6305.693} C_VEL
LIN {X 0,Y 495.87,Z 372.207,A -85,B 0,C 180,E1 -6308.148,E2 -6308.148} C_VEL
LIN {X 0,Y 495.865,Z 372.209,A -85,B 0,C 180,E1 -6311.444,E2 -6311.444} C_VEL
LIN {X 0,Y 495.787,Z 372.224,A -85,B 0,C 180,E1 -6314.782,E2 -6314.782} C_VEL
LIN {X 0,Y 495.784,Z 372.227,A -85,B 0,C 180,E1 -6317.318,E2 -6317.318} C_VEL
LIN {X 0,Y 495.768,Z 372.223,A -85,B 0,C 180,E1 -6319.89,E2 -6319.89} C_VEL
LIN {X 0,Y 495.757,Z 372.227,A -85,B 0,C 180,E1 -6322.861,E2 -6322.861} C_VEL
LIN {X 0,Y 495.796,Z 372.217,A -85,B 0,C 180,E1 -6326.067,E2 -6326.067} C_VEL
LIN {X 0,Y 495.768,Z 372.221,A -85,B 0,C 180,E1 -6328.814,E2 -6328.814} C_VEL
LIN {X 0,Y 495.755,Z 372.231,A -85,B 0,C 180,E1 -6331.726,E2 -6331.726} C_VEL
LIN {X 0,Y 495.772,Z 372.218,A -85,B 0,C 180,E1 -6334.695,E2 -6334.695} C_VEL
LIN {X 0,Y 495.728,Z 372.237,A -85,B 0,C 180,E1 -6337.561,E2 -6337.561} C_VEL
LIN {X 0,Y 495.763,Z 372.222,A -85,B 0,C 180,E1 -6340.7,E2 -6340.7} C_VEL
LIN {X 0,Y 495.731,Z 372.233,A -85,B 0,C 180,E1 -6343.695,E2 -6343.695} C_VEL
LIN {X 0,Y 495.724,Z 372.223,A -85,B 0,C 180,E1 -6346.305,E2 -6346.305} C_VEL
LIN {X 0,Y 495.776,Z 372.217,A -85,B 0,C 180,E1 -6349.301,E2 -6349.301} C_VEL
LIN {X 0,Y 495.728,Z 372.232,A -85,B 0,C 180,E1 -6352.438,E2 -6352.438} C_VEL
LIN {X 0,Y 495.781,Z 372.219,A -85,B 0,C 180,E1 -6355.457,E2 -6355.457} C_VEL
LIN {X 0,Y 495.756,Z 372.228,A -85,B 0,C 180,E1 -6358.364,E2 -6358.364} C_VEL
LIN {X 0,Y 495.761,Z 372.221,A -85,B 0,C 180,E1 -6360.763,E2 -6360.763} C_VEL
LIN {X 0,Y 495.1,Z 372.311,A -85,B 0,C 180,E1 -6361.442,E2 -6361.442} C_VEL
LIN {X 0,Y 492.238,Z 372.667,A -85,B 0,C 180,E1 -6362.545,E2 -6362.545} C_VEL
LIN {X 0,Y 489.828,Z 372.972,A -85,B 0,C 180,E1 -6363.433,E2 -6363.433} C_VEL
LIN {X 0,Y 488.811,Z 373.094,A -85,B 0,C 180,E1 -6364.12,E2 -6364.12} C_VEL
LIN {X 0,Y 488.739,Z 373.103,A -85,B 0,C 180,E1 -6364.352,E2 -6364.352} C_VEL
LIN {X 0,Y 488.718,Z 373.112,A -85,B 0,C 180,E1 -6367.153,E2 -6367.153} C_VEL
LIN {X 0,Y 488.725,Z 373.106,A -85,B 0,C 180,E1 -6369.811,E2 -6369.811} C_VEL
LIN {X 0,Y 488.731,Z 373.106,A -85,B 0,C 180,E1 -6372.423,E2 -6372.423} C_VEL
LIN {X 0,Y 488.758,Z 373.106,A -85,B 0,C 180,E1 -6374.999,E2 -6374.999} C_VEL
LIN {X 0,Y 488.802,Z 373.097,A -85,B 0,C 180,E1 -6378.387,E2 -6378.387} C_VEL
LIN {X 0,Y 488.814,Z 373.096,A -85,B 0,C 180,E1 -6381.733,E2 -6381.733} C_VEL
LIN {X 0,Y 488.855,Z 373.09,A -85,B 0,C 180,E1 -6384.224,E2 -6384.224} C_VEL
LIN {X 0,Y 488.959,Z 373.079,A -85,B 0,C 180,E1 -6387.528,E2 -6387.528} C_VEL
LIN {X 0,Y 488.951,Z 373.082,A -85,B 0,C 180,E1 -6390.823,E2 -6390.823} C_VEL
LIN {X 0,Y 488.959,Z 373.079,A -85,B 0,C 180,E1 -6392.471,E2 -6392.471} C_VEL
LIN {X 0,Y 488.855,Z 373.09,A -85,B 0,C 180,E1 -6395.775,E2 -6395.775} C_VEL
LIN {X 0,Y 488.814,Z 373.096,A -85,B 0,C 180,E1 -6398.266,E2 -6398.266} C_VEL
LIN {X 0,Y 488.802,Z 373.097,A -85,B 0,C 180,E1 -6401.612,E2 -6401.612} C_VEL
LIN {X 0,Y 488.757,Z 373.107,A -85,B 0,C 180,E1 -6405,E2 -6405} C_VEL
LIN {X 0,Y 488.75,Z 373.105,A -85,B 0,C 180,E1 -6408.442,E2 -6408.442} C_VEL
LIN {X 0,Y 488.703,Z 373.113,A -85,B 0,C 180,E1 -6411.07,E2 -6411.07} C_VEL
LIN {X 0,Y 488.689,Z 373.109,A -85,B 0,C 180,E1 -6413.745,E2 -6413.745} C_VEL
LIN {X 0,Y 488.794,Z 373.102,A -85,B 0,C 180,E1 -6416.945,E2 -6416.945} C_VEL
LIN {X 0,Y 488.713,Z 373.102,A -85,B 0,C 180,E1 -6420.365,E2 -6420.365} C_VEL
LIN {X 0,Y 488.73,Z 373.097,A -85,B 0,C 180,E1 -6423.484,E2 -6423.484} C_VEL
LIN {X 0,Y 488.683,Z 373.106,A -85,B 0,C 180,E1 -6426.356,E2 -6426.356} C_VEL
LIN {X 0,Y 488.736,Z 373.1,A -85,B 0,C 180,E1 -6429.25,E2 -6429.25} C_VEL
LIN {X 0,Y 488.705,Z 373.088,A -85,B 0,C 180,E1 -6431.6,E2 -6431.6} C_VEL
LIN {X 0,Y 488.705,Z 373.108,A -85,B 0,C 180,E1 -6434.801,E2 -6434.801} C_VEL
LIN {X 0,Y 488.688,Z 373.107,A -85,B 0,C 180,E1 -6437.475,E2 -6437.475} C_VEL
LIN {X 0,Y 488.723,Z 373.109,A -85,B 0,C 180,E1 -6440.749,E2 -6440.749} C_VEL
LIN {X 0,Y 488.678,Z 373.108,A -85,B 0,C 180,E1 -6443.869,E2 -6443.869} C_VEL
LIN {X 0,Y 488.732,Z 373.106,A -85,B 0,C 180,E1 -6446.877,E2 -6446.877} C_VEL
LIN {X 0,Y 488.727,Z 373.103,A -85,B 0,C 180,E1 -6449.782,E2 -6449.782} C_VEL
LIN {X 0,Y 488.791,Z 373.09,A -85,B 0,C 180,E1 -6453.055,E2 -6453.055} C_VEL
LIN {X 0,Y 488.686,Z 373.112,A -85,B 0,C 180,E1 -6456.255,E2 -6456.255} C_VEL
LIN {X 0,Y 488.738,Z 373.095,A -85,B 0,C 180,E1 -6459.176,E2 -6459.176} C_VEL
LIN {X 0,Y 488.752,Z 373.09,A -85,B 0,C 180,E1 -6461.628,E2 -6461.628} C_VEL
LIN {X 0,Y 488.755,Z 373.101,A -85,B 0,C 180,E1 -6465,E2 -6465} C_VEL
LIN {X 0,Y 488.823,Z 373.088,A -85,B 0,C 180,E1 -6468.388,E2 -6468.388} C_VEL
LIN {X 0,Y 488.811,Z 373.086,A -85,B 0,C 180,E1 -6471.734,E2 -6471.734} C_VEL
LIN {X 0,Y 488.849,Z 373.092,A -85,B 0,C 180,E1 -6474.225,E2 -6474.225} C_VEL
LIN {X 0,Y 488.956,Z 373.069,A -85,B 0,C 180,E1 -6477.529,E2 -6477.529} C_VEL
LIN {X 0,Y 488.949,Z 373.071,A -85,B 0,C 180,E1 -6480.824,E2 -6480.824} C_VEL
LIN {X 0,Y 488.956,Z 373.079,A -85,B 0,C 180,E1 -6482.472,E2 -6482.472} C_VEL
LIN {X 0,Y 488.85,Z 373.089,A -85,B 0,C 180,E1 -6485.776,E2 -6485.776} C_VEL
LIN {X 0,Y 488.812,Z 373.086,A -85,B 0,C 180,E1 -6488.267,E2 -6488.267} C_VEL
LIN {X 0,Y 488.8,Z 373.088,A -85,B 0,C 180,E1 -6491.613,E2 -6491.613} C_VEL
LIN {X 0,Y 488.757,Z 373.097,A -85,B 0,C 180,E1 -6495.001,E2 -6495.001} C_VEL
LIN {X 0,Y 488.75,Z 373.093,A -85,B 0,C 180,E1 -6498.443,E2 -6498.443} C_VEL
LIN {X 0,Y 488.702,Z 373.103,A -85,B 0,C 180,E1 -6501.071,E2 -6501.071} C_VEL
LIN {X 0,Y 488.69,Z 373.109,A -85,B 0,C 180,E1 -6503.746,E2 -6503.746} C_VEL
LIN {X 0,Y 488.795,Z 373.085,A -85,B 0,C 180,E1 -6506.946,E2 -6506.946} C_VEL
LIN {X 0,Y 488.716,Z 373.109,A -85,B 0,C 180,E1 -6510.366,E2 -6510.366} C_VEL
LIN {X 0,Y 488.733,Z 373.098,A -85,B 0,C 180,E1 -6513.485,E2 -6513.485} C_VEL
LIN {X 0,Y 488.687,Z 373.113,A -85,B 0,C 180,E1 -6516.357,E2 -6516.357} C_VEL
LIN {X 0,Y 488.74,Z 373.098,A -85,B 0,C 180,E1 -6519.251,E2 -6519.251} C_VEL
LIN {X 0,Y 488.73,Z 373.104,A -85,B 0,C 180,E1 -6522.522,E2 -6522.522} C_VEL
LIN {X 0,Y 488.71,Z 373.104,A -85,B 0,C 180,E1 -6525.199,E2 -6525.199} C_VEL
LIN {X 0,Y 488.707,Z 373.099,A -85,B 0,C 180,E1 -6528.401,E2 -6528.401} C_VEL
LIN {X 0,Y 488.704,Z 373.105,A -85,B 0,C 180,E1 -6530.948,E2 -6530.948} C_VEL
LIN {X 0,Y 488.685,Z 373.108,A -85,B 0,C 180,E1 -6533.869,E2 -6533.869} C_VEL
LIN {X 0,Y 488.739,Z 373.1,A -85,B 0,C 180,E1 -6536.878,E2 -6536.878} C_VEL
LIN {X 0,Y 488.735,Z 373.106,A -85,B 0,C 180,E1 -6539.782,E2 -6539.782} C_VEL
LIN {X 0,Y 488.797,Z 373.233,A -85,B 0,C 180,E1 -6543.056,E2 -6543.056} C_VEL
LIN {X 0,Y 490.295,Z 381.672,A -85,B 0,C 180,E1 -6545.042,E2 -6545.042} C_VEL
LIN {X 0,Y 490.099,Z 390.225,A -85,B 0,C 180,E1 -6546.901,E2 -6546.901} C_VEL
LIN {X 0,Y 489.588,Z 404.222,A -85,B 0,C 180,E1 -6549.848,E2 -6549.848} C_VEL
LIN {X 0,Y 489.092,Z 418.68,A -85,B 0,C 180,E1 -6552.868,E2 -6552.868} C_VEL
LIN {X 0,Y 488.996,Z 422.813,A -85,B 0,C 180,E1 -6553.714,E2 -6553.714} C_VEL
LIN {X 0,Y 490.675,Z 433.059,A -85,B 0,C 180,E1 -6553.954,E2 -6553.954} C_VEL
LIN {X 0,Y 491.704,Z 440.374,A -85,B 0,C 180,E1 -6554.096,E2 -6554.096} C_VEL
LIN {X 0,Y 491.151,Z 527.637,A -85,B 0,C 180,E1 -6555.393,E2 -6555.393} C_VEL
LIN {X 0,Y 490.938,Z 537.551,A -85,B 0,C 180,E1 -6555.624,E2 -6555.624} C_VEL
LIN {X 0,Y 490.689,Z 547.539,A -85,B 0,C 180,E1 -6555.961,E2 -6555.961} C_VEL
LIN {X 0,Y 490.334,Z 557.897,A -85,B 0,C 180,E1 -6556.426,E2 -6556.426} C_VEL
LIN {X 0,Y 490.028,Z 567.323,A -85,B 0,C 180,E1 -6556.964,E2 -6556.964} C_VEL
LIN {X 0,Y 489.698,Z 576.051,A -85,B 0,C 180,E1 -6557.569,E2 -6557.569} C_VEL
LIN {X 0,Y 489.405,Z 584.782,A -85,B 0,C 180,E1 -6558.297,E2 -6558.297} C_VEL
LIN {X 0,Y 489.122,Z 592.206,A -85,B 0,C 180,E1 -6559.025,E2 -6559.025} C_VEL
LIN {X 0,Y 488.718,Z 601.003,A -85,B 0,C 180,E1 -6560.063,E2 -6560.063} C_VEL
LIN {X 0,Y 488.518,Z 606.995,A -85,B 0,C 180,E1 -6560.895,E2 -6560.895} C_VEL
LIN {X 0,Y 488.318,Z 613.306,A -85,B 0,C 180,E1 -6561.934,E2 -6561.934} C_VEL
LIN {X 0,Y 488.143,Z 618.578,A -85,B 0,C 180,E1 -6562.971,E2 -6562.971} C_VEL
LIN {X 0,Y 488.037,Z 623.669,A -85,B 0,C 180,E1 -6564.215,E2 -6564.215} C_VEL
LIN {X 0,Y 487.921,Z 627.628,A -85,B 0,C 180,E1 -6565.456,E2 -6565.456} C_VEL
LIN {X 0,Y 487.965,Z 630.559,A -85,B 0,C 180,E1 -6566.698,E2 -6566.698} C_VEL
LIN {X 0,Y 487.909,Z 632.055,A -85,B 0,C 180,E1 -6567.524,E2 -6567.524} C_VEL
LIN {X 0,Y 487.834,Z 633.571,A -85,B 0,C 180,E1 -6569.175,E2 -6569.175} C_VEL
LIN {X 0,Y 487.819,Z 633.849,A -85,B 0,C 180,E1 -6570,E2 -6570} C_VEL
LIN {X 0,Y 487.891,Z 632.979,A -85,B 0,C 180,E1 -6571.651,E2 -6571.651} C_VEL
LIN {X 0,Y 487.909,Z 632.054,A -85,B 0,C 180,E1 -6572.477,E2 -6572.477} C_VEL
LIN {X 0,Y 487.928,Z 628.714,A -85,B 0,C 180,E1 -6574.13,E2 -6574.13} C_VEL
LIN {X 0,Y 488.022,Z 625.094,A -85,B 0,C 180,E1 -6575.371,E2 -6575.371} C_VEL
LIN {X 0,Y 488.069,Z 620.365,A -85,B 0,C 180,E1 -6576.615,E2 -6576.615} C_VEL
LIN {X 0,Y 488.247,Z 614.395,A -85,B 0,C 180,E1 -6577.86,E2 -6577.86} C_VEL
LIN {X 0,Y 488.458,Z 608.304,A -85,B 0,C 180,E1 -6578.898,E2 -6578.898} C_VEL
LIN {X 0,Y 488.679,Z 602.561,A -85,B 0,C 180,E1 -6579.729,E2 -6579.729} C_VEL
LIN {X 0,Y 488.898,Z 595.902,A -85,B 0,C 180,E1 -6580.561,E2 -6580.561} C_VEL
LIN {X 0,Y 489.251,Z 588.073,A -85,B 0,C 180,E1 -6581.392,E2 -6581.392} C_VEL
LIN {X 0,Y 489.621,Z 579.987,A -85,B 0,C 180,E1 -6582.118,E2 -6582.118} C_VEL
LIN {X 0,Y 489.94,Z 570.547,A -85,B 0,C 180,E1 -6582.825,E2 -6582.825} C_VEL
LIN {X 0,Y 490.227,Z 561.826,A -85,B 0,C 180,E1 -6583.366,E2 -6583.366} C_VEL
LIN {X 0,Y 490.581,Z 551.316,A -85,B 0,C 180,E1 -6583.884,E2 -6583.884} C_VEL
LIN {X 0,Y 490.843,Z 540.979,A -85,B 0,C 180,E1 -6584.273,E2 -6584.273} C_VEL
LIN {X 0,Y 491.135,Z 530.256,A -85,B 0,C 180,E1 -6584.555,E2 -6584.555} C_VEL
LIN {X 0,Y 491.321,Z 507.477,A -85,B 0,C 180,E1 -6584.92,E2 -6584.92} C_VEL
LIN {X 0,Y 491.543,Z 438.078,A -85,B 0,C 180,E1 -6585.943,E2 -6585.943} C_VEL
LIN {X 0,Y 489.035,Z 422.936,A -85,B 0,C 180,E1 -6586.275,E2 -6586.275} C_VEL
LIN {X 0,Y 489.018,Z 422.128,A -85,B 0,C 180,E1 -6586.383,E2 -6586.383} C_VEL
LIN {X 0,Y 489.445,Z 408.472,A -85,B 0,C 180,E1 -6589.285,E2 -6589.285} C_VEL
LIN {X 0,Y 489.951,Z 393.824,A -85,B 0,C 180,E1 -6592.341,E2 -6592.341} C_VEL
LIN {X 0,Y 490.377,Z 383.508,A -85,B 0,C 180,E1 -6594.558,E2 -6594.558} C_VEL
LIN {X 0,Y 489.552,Z 377.317,A -85,B 0,C 180,E1 -6595.967,E2 -6595.967} C_VEL
LIN {X 0,Y 488.778,Z 373.229,A -85,B 0,C 180,E1 -6596.939,E2 -6596.939} C_VEL
LIN {X 0,Y 488.737,Z 373.106,A -85,B 0,C 180,E1 -6600.218,E2 -6600.218} C_VEL
LIN {X 0,Y 488.738,Z 373.102,A -85,B 0,C 180,E1 -6603.484,E2 -6603.484} C_VEL
LIN {X 0,Y 488.691,Z 373.109,A -85,B 0,C 180,E1 -6606.355,E2 -6606.355} C_VEL
LIN {X 0,Y 488.704,Z 373.106,A -85,B 0,C 180,E1 -6609.254,E2 -6609.254} C_VEL
LIN {X 0,Y 488.71,Z 373.098,A -85,B 0,C 180,E1 -6611.6,E2 -6611.6} C_VEL
LIN {X 0,Y 488.713,Z 373.104,A -85,B 0,C 180,E1 -6614.801,E2 -6614.801} C_VEL
LIN {X 0,Y 488.733,Z 373.104,A -85,B 0,C 180,E1 -6617.478,E2 -6617.478} C_VEL
LIN {X 0,Y 488.743,Z 373.098,A -85,B 0,C 180,E1 -6620.749,E2 -6620.749} C_VEL
LIN {X 0,Y 488.684,Z 373.114,A -85,B 0,C 180,E1 -6623.868,E2 -6623.868} C_VEL
LIN {X 0,Y 488.739,Z 373.096,A -85,B 0,C 180,E1 -6626.877,E2 -6626.877} C_VEL
LIN {X 0,Y 488.734,Z 373.109,A -85,B 0,C 180,E1 -6629.781,E2 -6629.781} C_VEL
LIN {X 0,Y 488.792,Z 373.086,A -85,B 0,C 180,E1 -6633.056,E2 -6633.056} C_VEL
LIN {X 0,Y 488.693,Z 373.109,A -85,B 0,C 180,E1 -6636.254,E2 -6636.254} C_VEL
LIN {X 0,Y 488.745,Z 373.099,A -85,B 0,C 180,E1 -6639.175,E2 -6639.175} C_VEL
LIN {X 0,Y 488.733,Z 373.095,A -85,B 0,C 180,E1 -6642.423,E2 -6642.423} C_VEL
LIN {X 0,Y 488.761,Z 373.097,A -85,B 0,C 180,E1 -6644.999,E2 -6644.999} C_VEL
LIN {X 0,Y 488.804,Z 373.088,A -85,B 0,C 180,E1 -6648.387,E2 -6648.387} C_VEL
LIN {X 0,Y 488.815,Z 373.085,A -85,B 0,C 180,E1 -6651.733,E2 -6651.733} C_VEL
LIN {X 0,Y 488.853,Z 373.088,A -85,B 0,C 180,E1 -6654.224,E2 -6654.224} C_VEL
LIN {X 0,Y 488.959,Z 373.079,A -85,B 0,C 180,E1 -6657.528,E2 -6657.528} C_VEL
LIN {X 0,Y 488.967,Z 373.062,A -85,B 0,C 180,E1 -6660,E2 -6660} C_VEL
LIN {X 0,Y 488.959,Z 373.069,A -85,B 0,C 180,E1 -6662.471,E2 -6662.471} C_VEL
LIN {X 0,Y 488.852,Z 373.092,A -85,B 0,C 180,E1 -6665.775,E2 -6665.775} C_VEL
LIN {X 0,Y 488.814,Z 373.085,A -85,B 0,C 180,E1 -6668.266,E2 -6668.266} C_VEL
LIN {X 0,Y 488.826,Z 373.088,A -85,B 0,C 180,E1 -6671.611,E2 -6671.611} C_VEL
LIN {X 0,Y 488.759,Z 373.101,A -85,B 0,C 180,E1 -6675,E2 -6675} C_VEL
LIN {X 0,Y 488.751,Z 373.09,A -85,B 0,C 180,E1 -6678.442,E2 -6678.442} C_VEL
LIN {X 0,Y 488.703,Z 373.102,A -85,B 0,C 180,E1 -6681.07,E2 -6681.07} C_VEL
LIN {X 0,Y 488.689,Z 373.112,A -85,B 0,C 180,E1 -6683.745,E2 -6683.745} C_VEL
LIN {X 0,Y 488.795,Z 373.09,A -85,B 0,C 180,E1 -6686.945,E2 -6686.945} C_VEL
LIN {X 0,Y 488.706,Z 373.105,A -85,B 0,C 180,E1 -6690.363,E2 -6690.363} C_VEL
LIN {X 0,Y 488.732,Z 373.102,A -85,B 0,C 180,E1 -6693.484,E2 -6693.484} C_VEL
LIN {X 0,Y 488.685,Z 373.107,A -85,B 0,C 180,E1 -6696.355,E2 -6696.355} C_VEL
LIN {X 0,Y 488.697,Z 373.112,A -85,B 0,C 180,E1 -6699.254,E2 -6699.254} C_VEL
LIN {X 0,Y 488.72,Z 373.108,A -85,B 0,C 180,E1 -6701.602,E2 -6701.602} C_VEL
LIN {X 0,Y 488.708,Z 373.107,A -85,B 0,C 180,E1 -6704.801,E2 -6704.801} C_VEL
LIN {X 0,Y 488.687,Z 373.093,A -85,B 0,C 180,E1 -6707.474,E2 -6707.474} C_VEL
LIN {X 0,Y 488.729,Z 373.102,A -85,B 0,C 180,E1 -6709.677,E2 -6709.677} C_VEL
LIN {X 0,Y 488.676,Z 373.11,A -85,B 0,C 180,E1 -6712.278,E2 -6712.278} C_VEL
LIN {X 0,Y 488.725,Z 373.098,A -85,B 0,C 180,E1 -6715.051,E2 -6715.051} C_VEL
LIN {X 0,Y 488.703,Z 373.107,A -85,B 0,C 180,E1 -6718.045,E2 -6718.045} C_VEL
LIN {X 0,Y 488.729,Z 373.099,A -85,B 0,C 180,E1 -6720.76,E2 -6720.76} C_VEL
LIN {X 0,Y 488.753,Z 373.105,A -85,B 0,C 180,E1 -6723.528,E2 -6723.528} C_VEL
LIN {X 0,Y 488.739,Z 373.103,A -85,B 0,C 180,E1 -6724.352,E2 -6724.352} C_VEL
LIN {X 0,Y 488.095,Z 373.189,A -85,B 0,C 180,E1 -6725.04,E2 -6725.04} C_VEL
LIN {X 0,Y 485.226,Z 373.545,A -85,B 0,C 180,E1 -6726.156,E2 -6726.156} C_VEL
LIN {X 0,Y 482.779,Z 373.851,A -85,B 0,C 180,E1 -6727.056,E2 -6727.056} C_VEL
LIN {X 0,Y 481.722,Z 373.979,A -85,B 0,C 180,E1 -6727.751,E2 -6727.751} C_VEL
LIN {X 0,Y 481.633,Z 373.989,A -85,B 0,C 180,E1 -6727.987,E2 -6727.987} C_VEL
LIN {X 0,Y 481.705,Z 373.981,A -85,B 0,C 180,E1 -6730.393,E2 -6730.393} C_VEL
LIN {X 0,Y 481.688,Z 373.987,A -85,B 0,C 180,E1 -6733.034,E2 -6733.034} C_VEL
LIN {X 0,Y 481.686,Z 373.985,A -85,B 0,C 180,E1 -6735.639,E2 -6735.639} C_VEL
LIN {X 0,Y 481.748,Z 373.975,A -85,B 0,C 180,E1 -6738.215,E2 -6738.215} C_VEL
LIN {X 0,Y 481.759,Z 373.976,A -85,B 0,C 180,E1 -6741.612,E2 -6741.612} C_VEL
LIN {X 0,Y 481.816,Z 373.967,A -85,B 0,C 180,E1 -6744.139,E2 -6744.139} C_VEL
LIN {X 0,Y 481.925,Z 373.956,A -85,B 0,C 180,E1 -6747.492,E2 -6747.492} C_VEL
LIN {X 0,Y 481.902,Z 373.96,A -85,B 0,C 180,E1 -6750.835,E2 -6750.835} C_VEL
LIN {X 0,Y 481.925,Z 373.955,A -85,B 0,C 180,E1 -6752.507,E2 -6752.507} C_VEL
LIN {X 0,Y 481.816,Z 373.967,A -85,B 0,C 180,E1 -6755.86,E2 -6755.86} C_VEL
LIN {X 0,Y 481.759,Z 373.976,A -85,B 0,C 180,E1 -6758.388,E2 -6758.388} C_VEL
LIN {X 0,Y 481.747,Z 373.975,A -85,B 0,C 180,E1 -6761.785,E2 -6761.785} C_VEL
LIN {X 0,Y 481.738,Z 373.98,A -85,B 0,C 180,E1 -6765.224,E2 -6765.224} C_VEL
LIN {X 0,Y 481.708,Z 373.985,A -85,B 0,C 180,E1 -6768.721,E2 -6768.721} C_VEL
LIN {X 0,Y 481.642,Z 373.989,A -85,B 0,C 180,E1 -6771.394,E2 -6771.394} C_VEL
LIN {X 0,Y 481.672,Z 373.984,A -85,B 0,C 180,E1 -6774.113,E2 -6774.113} C_VEL
LIN {X 0,Y 481.747,Z 373.977,A -85,B 0,C 180,E1 -6777.14,E2 -6777.14} C_VEL
LIN {X 0,Y 481.683,Z 373.974,A -85,B 0,C 180,E1 -6779.74,E2 -6779.74} C_VEL
LIN {X 0,Y 481.667,Z 373.987,A -85,B 0,C 180,E1 -6782.674,E2 -6782.674} C_VEL
LIN {X 0,Y 481.637,Z 373.98,A -85,B 0,C 180,E1 -6785.709,E2 -6785.709} C_VEL
LIN {X 0,Y 481.708,Z 373.975,A -85,B 0,C 180,E1 -6789.354,E2 -6789.354} C_VEL
LIN {X 0,Y 481.642,Z 373.967,A -85,B 0,C 180,E1 -6792.16,E2 -6792.16} C_VEL
LIN {X 0,Y 481.653,Z 373.983,A -85,B 0,C 180,E1 -6795.543,E2 -6795.543} C_VEL
LIN {X 0,Y 481.655,Z 373.984,A -85,B 0,C 180,E1 -6798.086,E2 -6798.086} C_VEL
LIN {X 0,Y 481.664,Z 373.985,A -85,B 0,C 180,E1 -6801.141,E2 -6801.141} C_VEL
LIN {X 0,Y 481.661,Z 373.98,A -85,B 0,C 180,E1 -6804.795,E2 -6804.795} C_VEL
LIN {X 0,Y 481.666,Z 373.982,A -85,B 0,C 180,E1 -6807.326,E2 -6807.326} C_VEL
LIN {X 0,Y 481.681,Z 373.985,A -85,B 0,C 180,E1 -6810.26,E2 -6810.26} C_VEL
LIN {X 0,Y 481.745,Z 373.967,A -85,B 0,C 180,E1 -6813.113,E2 -6813.113} C_VEL
LIN {X 0,Y 481.67,Z 373.982,A -85,B 0,C 180,E1 -6815.887,E2 -6815.887} C_VEL
LIN {X 0,Y 481.695,Z 373.974,A -85,B 0,C 180,E1 -6819.028,E2 -6819.028} C_VEL
LIN {X 0,Y 481.701,Z 373.972,A -85,B 0,C 180,E1 -6822.159,E2 -6822.159} C_VEL
LIN {X 0,Y 481.735,Z 373.978,A -85,B 0,C 180,E1 -6824.776,E2 -6824.776} C_VEL
LIN {X 0,Y 481.788,Z 373.968,A -85,B 0,C 180,E1 -6828.217,E2 -6828.217} C_VEL
LIN {X 0,Y 481.756,Z 373.964,A -85,B 0,C 180,E1 -6831.612,E2 -6831.612} C_VEL
LIN {X 0,Y 481.81,Z 373.968,A -85,B 0,C 180,E1 -6834.14,E2 -6834.14} C_VEL
LIN {X 0,Y 481.923,Z 373.945,A -85,B 0,C 180,E1 -6837.493,E2 -6837.493} C_VEL
LIN {X 0,Y 481.9,Z 373.948,A -85,B 0,C 180,E1 -6840.836,E2 -6840.836} C_VEL
LIN {X 0,Y 481.923,Z 373.955,A -85,B 0,C 180,E1 -6842.508,E2 -6842.508} C_VEL
LIN {X 0,Y 481.811,Z 373.966,A -85,B 0,C 180,E1 -6845.861,E2 -6845.861} C_VEL
LIN {X 0,Y 481.757,Z 373.962,A -85,B 0,C 180,E1 -6848.389,E2 -6848.389} C_VEL
LIN {X 0,Y 481.745,Z 373.968,A -85,B 0,C 180,E1 -6851.786,E2 -6851.786} C_VEL
LIN {X 0,Y 481.737,Z 373.971,A -85,B 0,C 180,E1 -6855.225,E2 -6855.225} C_VEL
LIN {X 0,Y 481.708,Z 373.968,A -85,B 0,C 180,E1 -6858.722,E2 -6858.722} C_VEL
LIN {X 0,Y 481.642,Z 373.983,A -85,B 0,C 180,E1 -6861.395,E2 -6861.395} C_VEL
LIN {X 0,Y 481.673,Z 373.986,A -85,B 0,C 180,E1 -6864.114,E2 -6864.114} C_VEL
LIN {X 0,Y 481.748,Z 373.962,A -85,B 0,C 180,E1 -6867.141,E2 -6867.141} C_VEL
LIN {X 0,Y 481.685,Z 373.982,A -85,B 0,C 180,E1 -6869.741,E2 -6869.741} C_VEL
LIN {X 0,Y 481.67,Z 373.978,A -85,B 0,C 180,E1 -6872.675,E2 -6872.675} C_VEL
LIN {X 0,Y 481.64,Z 373.985,A -85,B 0,C 180,E1 -6875.71,E2 -6875.71} C_VEL
LIN {X 0,Y 481.712,Z 373.974,A -85,B 0,C 180,E1 -6879.355,E2 -6879.355} C_VEL
LIN {X 0,Y 481.672,Z 373.988,A -85,B 0,C 180,E1 -6882.159,E2 -6882.159} C_VEL
LIN {X 0,Y 481.658,Z 373.985,A -85,B 0,C 180,E1 -6884.458,E2 -6884.458} C_VEL
LIN {X 0,Y 481.647,Z 373.987,A -85,B 0,C 180,E1 -6887.84,E2 -6887.84} C_VEL
LIN {X 0,Y 481.68,Z 373.981,A -85,B 0,C 180,E1 -6890.652,E2 -6890.652} C_VEL
LIN {X 0,Y 481.632,Z 373.987,A -85,B 0,C 180,E1 -6893.376,E2 -6893.376} C_VEL
LIN {X 0,Y 481.71,Z 373.979,A -85,B 0,C 180,E1 -6896.331,E2 -6896.331} C_VEL
LIN {X 0,Y 481.659,Z 373.989,A -85,B 0,C 180,E1 -6899.416,E2 -6899.416} C_VEL
LIN {X 0,Y 481.707,Z 373.985,A -85,B 0,C 180,E1 -6902.56,E2 -6902.56} C_VEL
LIN {X 0,Y 481.753,Z 374.114,A -85,B 0,C 180,E1 -6902.86,E2 -6902.86} C_VEL
LIN {X 0,Y 483.376,Z 383.364,A -85,B 0,C 180,E1 -6905.062,E2 -6905.062} C_VEL
LIN {X 0,Y 482.976,Z 395.773,A -85,B 0,C 180,E1 -6907.77,E2 -6907.77} C_VEL
LIN {X 0,Y 482.382,Z 410.458,A -85,B 0,C 180,E1 -6910.909,E2 -6910.909} C_VEL
LIN {X 0,Y 481.992,Z 422.624,A -85,B 0,C 180,E1 -6913.471,E2 -6913.471} C_VEL
LIN {X 0,Y 483.645,Z 432.336,A -85,B 0,C 180,E1 -6913.706,E2 -6913.706} C_VEL
LIN {X 0,Y 484.878,Z 440.61,A -85,B 0,C 180,E1 -6913.873,E2 -6913.873} C_VEL
LIN {X 0,Y 484.3,Z 527.443,A -85,B 0,C 180,E1 -6915.181,E2 -6915.181} C_VEL
LIN {X 0,Y 484.083,Z 537.357,A -85,B 0,C 180,E1 -6915.416,E2 -6915.416} C_VEL
LIN {X 0,Y 483.797,Z 547.344,A -85,B 0,C 180,E1 -6915.757,E2 -6915.757} C_VEL
LIN {X 0,Y 483.438,Z 557.702,A -85,B 0,C 180,E1 -6916.229,E2 -6916.229} C_VEL
LIN {X 0,Y 483.086,Z 566.853,A -85,B 0,C 180,E1 -6916.755,E2 -6916.755} C_VEL
LIN {X 0,Y 482.695,Z 576.668,A -85,B 0,C 180,E1 -6917.452,E2 -6917.452} C_VEL
LIN {X 0,Y 482.421,Z 584.586,A -85,B 0,C 180,E1 -6918.125,E2 -6918.125} C_VEL
LIN {X 0,Y 482.138,Z 592.011,A -85,B 0,C 180,E1 -6918.864,E2 -6918.864} C_VEL
LIN {X 0,Y 481.687,Z 600.807,A -85,B 0,C 180,E1 -6919.917,E2 -6919.917} C_VEL
LIN {X 0,Y 481.46,Z 606.799,A -85,B 0,C 180,E1 -6920.76,E2 -6920.76} C_VEL
LIN {X 0,Y 481.248,Z 613.11,A -85,B 0,C 180,E1 -6921.814,E2 -6921.814} C_VEL
LIN {X 0,Y 481.079,Z 618.383,A -85,B 0,C 180,E1 -6922.867,E2 -6922.867} C_VEL
LIN {X 0,Y 480.94,Z 623.474,A -85,B 0,C 180,E1 -6924.129,E2 -6924.129} C_VEL
LIN {X 0,Y 480.84,Z 627.433,A -85,B 0,C 180,E1 -6925.389,E2 -6925.389} C_VEL
LIN {X 0,Y 480.888,Z 630.364,A -85,B 0,C 180,E1 -6926.649,E2 -6926.649} C_VEL
LIN {X 0,Y 480.823,Z 631.86,A -85,B 0,C 180,E1 -6927.487,E2 -6927.487} C_VEL
LIN {X 0,Y 480.76,Z 633.377,A -85,B 0,C 180,E1 -6929.163,E2 -6929.163} C_VEL
LIN {X 0,Y 480.743,Z 633.654,A -85,B 0,C 180,E1 -6930,E2 -6930} C_VEL
LIN {X 0,Y 480.792,Z 632.784,A -85,B 0,C 180,E1 -6931.676,E2 -6931.676} C_VEL
LIN {X 0,Y 480.823,Z 631.859,A -85,B 0,C 180,E1 -6932.513,E2 -6932.513} C_VEL
LIN {X 0,Y 480.889,Z 630.364,A -85,B 0,C 180,E1 -6933.352,E2 -6933.352} C_VEL
LIN {X 0,Y 480.899,Z 626.309,A -85,B 0,C 180,E1 -6935.031,E2 -6935.031} C_VEL
LIN {X 0,Y 480.951,Z 621.286,A -85,B 0,C 180,E1 -6936.45,E2 -6936.45} C_VEL
LIN {X 0,Y 481.154,Z 615.292,A -85,B 0,C 180,E1 -6937.765,E2 -6937.765} C_VEL
LIN {X 0,Y 481.375,Z 609.42,A -85,B 0,C 180,E1 -6938.818,E2 -6938.818} C_VEL
LIN {X 0,Y 481.579,Z 603.926,A -85,B 0,C 180,E1 -6939.662,E2 -6939.662} C_VEL
LIN {X 0,Y 481.89,Z 595.706,A -85,B 0,C 180,E1 -6940.717,E2 -6940.717} C_VEL
LIN {X 0,Y 482.271,Z 587.877,A -85,B 0,C 180,E1 -6941.559,E2 -6941.559} C_VEL
LIN {X 0,Y 482.648,Z 579.791,A -85,B 0,C 180,E1 -6942.296,E2 -6942.296} C_VEL
LIN {X 0,Y 482.94,Z 571.94,A -85,B 0,C 180,E1 -6942.907,E2 -6942.907} C_VEL
LIN {X 0,Y 483.306,Z 561.63,A -85,B 0,C 180,E1 -6943.561,E2 -6943.561} C_VEL
LIN {X 0,Y 483.693,Z 551.121,A -85,B 0,C 180,E1 -6944.086,E2 -6944.086} C_VEL
LIN {X 0,Y 483.953,Z 540.783,A -85,B 0,C 180,E1 -6944.481,E2 -6944.481} C_VEL
LIN {X 0,Y 484.275,Z 530.062,A -85,B 0,C 180,E1 -6944.766,E2 -6944.766} C_VEL
LIN {X 0,Y 484.455,Z 507.282,A -85,B 0,C 180,E1 -6945.137,E2 -6945.137} C_VEL
LIN {X 0,Y 484.736,Z 439.031,A -85,B 0,C 180,E1 -6946.156,E2 -6946.156} C_VEL
LIN {X 0,Y 482.008,Z 422.747,A -85,B 0,C 180,E1 -6946.519,E2 -6946.519} C_VEL
LIN {X 0,Y 481.989,Z 421.932,A -85,B 0,C 180,E1 -6946.628,E2 -6946.628} C_VEL
LIN {X 0,Y 482.491,Z 408.325,A -85,B 0,C 180,E1 -6949.574,E2 -6949.574} C_VEL
LIN {X 0,Y 483.02,Z 393.686,A -85,B 0,C 180,E1 -6952.68,E2 -6952.68} C_VEL
LIN {X 0,Y 483.359,Z 383.367,A -85,B 0,C 180,E1 -6954.939,E2 -6954.939} C_VEL
LIN {X 0,Y 481.726,Z 374.091,A -85,B 0,C 180,E1 -6957.162,E2 -6957.162} C_VEL
LIN {X 0,Y 481.691,Z 373.983,A -85,B 0,C 180,E1 -6959.74,E2 -6959.74} C_VEL
LIN {X 0,Y 481.675,Z 373.982,A -85,B 0,C 180,E1 -6962.674,E2 -6962.674} C_VEL
LIN {X 0,Y 481.645,Z 373.985,A -85,B 0,C 180,E1 -6965.709,E2 -6965.709} C_VEL
LIN {X 0,Y 481.673,Z 373.981,A -85,B 0,C 180,E1 -6968.859,E2 -6968.859} C_VEL
LIN {X 0,Y 481.655,Z 373.981,A -85,B 0,C 180,E1 -6971.913,E2 -6971.913} C_VEL
LIN {X 0,Y 481.661,Z 373.984,A -85,B 0,C 180,E1 -6974.457,E2 -6974.457} C_VEL
LIN {X 0,Y 481.69,Z 373.979,A -85,B 0,C 180,E1 -6976.845,E2 -6976.845} C_VEL
LIN {X 0,Y 481.69,Z 373.98,A -85,B 0,C 180,E1 -6980.06,E2 -6980.06} C_VEL
LIN {X 0,Y 481.629,Z 373.988,A -85,B 0,C 180,E1 -6983.253,E2 -6983.253} C_VEL
LIN {X 0,Y 481.71,Z 373.974,A -85,B 0,C 180,E1 -6986.33,E2 -6986.33} C_VEL
LIN {X 0,Y 481.659,Z 373.986,A -85,B 0,C 180,E1 -6989.415,E2 -6989.415} C_VEL
LIN {X 0,Y 481.701,Z 373.972,A -85,B 0,C 180,E1 -6992.168,E2 -6992.168} C_VEL
LIN {X 0,Y 481.718,Z 373.971,A -85,B 0,C 180,E1 -6994.969,E2 -6994.969} C_VEL
LIN {X 0,Y 481.653,Z 373.99,A -85,B 0,C 180,E1 -6997.704,E2 -6997.704} C_VEL
LIN {X 0,Y 481.705,Z 373.968,A -85,B 0,C 180,E1 -7000.393,E2 -7000.393} C_VEL
LIN {X 0,Y 481.69,Z 373.971,A -85,B 0,C 180,E1 -7003.033,E2 -7003.033} C_VEL
LIN {X 0,Y 481.689,Z 373.984,A -85,B 0,C 180,E1 -7005.638,E2 -7005.638} C_VEL
LIN {X 0,Y 481.749,Z 373.968,A -85,B 0,C 180,E1 -7008.215,E2 -7008.215} C_VEL
LIN {X 0,Y 481.761,Z 373.961,A -85,B 0,C 180,E1 -7011.611,E2 -7011.611} C_VEL
LIN {X 0,Y 481.814,Z 373.966,A -85,B 0,C 180,E1 -7014.139,E2 -7014.139} C_VEL
LIN {X 0,Y 481.926,Z 373.955,A -85,B 0,C 180,E1 -7017.492,E2 -7017.492} C_VEL
LIN {X 0,Y 481.938,Z 373.936,A -85,B 0,C 180,E1 -7020,E2 -7020} C_VEL
LIN {X 0,Y 481.926,Z 373.945,A -85,B 0,C 180,E1 -7022.507,E2 -7022.507} C_VEL
LIN {X 0,Y 481.813,Z 373.968,A -85,B 0,C 180,E1 -7025.86,E2 -7025.86} C_VEL
LIN {X 0,Y 481.76,Z 373.963,A -85,B 0,C 180,E1 -7028.388,E2 -7028.388} C_VEL
LIN {X 0,Y 481.792,Z 373.967,A -85,B 0,C 180,E1 -7031.783,E2 -7031.783} C_VEL
LIN {X 0,Y 481.739,Z 373.977,A -85,B 0,C 180,E1 -7035.224,E2 -7035.224} C_VEL
LIN {X 0,Y 481.708,Z 373.967,A -85,B 0,C 180,E1 -7038.721,E2 -7038.721} C_VEL
LIN {X 0,Y 481.642,Z 373.986,A -85,B 0,C 180,E1 -7041.394,E2 -7041.394} C_VEL
LIN {X 0,Y 481.673,Z 373.982,A -85,B 0,C 180,E1 -7044.113,E2 -7044.113} C_VEL
LIN {X 0,Y 481.748,Z 373.969,A -85,B 0,C 180,E1 -7047.14,E2 -7047.14} C_VEL
LIN {X 0,Y 481.675,Z 373.986,A -85,B 0,C 180,E1 -7049.741,E2 -7049.741} C_VEL
LIN {X 0,Y 481.669,Z 373.982,A -85,B 0,C 180,E1 -7052.674,E2 -7052.674} C_VEL
LIN {X 0,Y 481.638,Z 373.989,A -85,B 0,C 180,E1 -7055.709,E2 -7055.709} C_VEL
LIN {X 0,Y 481.667,Z 373.985,A -85,B 0,C 180,E1 -7058.859,E2 -7058.859} C_VEL
LIN {X 0,Y 481.658,Z 373.984,A -85,B 0,C 180,E1 -7061.914,E2 -7061.914} C_VEL
LIN {X 0,Y 481.656,Z 373.983,A -85,B 0,C 180,E1 -7064.457,E2 -7064.457} C_VEL
LIN {X 0,Y 481.644,Z 373.967,A -85,B 0,C 180,E1 -7067.839,E2 -7067.839} C_VEL
LIN {X 0,Y 481.71,Z 373.975,A -85,B 0,C 180,E1 -7070.646,E2 -7070.646} C_VEL
LIN {X 0,Y 481.639,Z 373.98,A -85,B 0,C 180,E1 -7074.291,E2 -7074.291} C_VEL
LIN {X 0,Y 481.669,Z 373.986,A -85,B 0,C 180,E1 -7077.326,E2 -7077.326} C_VEL
LIN {X 0,Y 481.685,Z 373.974,A -85,B 0,C 180,E1 -7080.259,E2 -7080.259} C_VEL
LIN {X 0,Y 481.742,Z 373.981,A -85,B 0,C 180,E1 -7083.112,E2 -7083.112} C_VEL
LIN {X 0,Y 481.674,Z 373.984,A -85,B 0,C 180,E1 -7085.887,E2 -7085.887} C_VEL
LIN {X 0,Y 481.633,Z 373.989,A -85,B 0,C 180,E1 -7087.987,E2 -7087.987} C_VEL
LIN {X 0,Y 480.966,Z 374.075,A -85,B 0,C 180,E1 -7088.685,E2 -7088.685} C_VEL
LIN {X 0,Y 478.139,Z 374.427,A -85,B 0,C 180,E1 -7089.819,E2 -7089.819} C_VEL
LIN {X 0,Y 475.754,Z 374.726,A -85,B 0,C 180,E1 -7090.733,E2 -7090.733} C_VEL
LIN {X 0,Y 474.734,Z 374.852,A -85,B 0,C 180,E1 -7091.439,E2 -7091.439} C_VEL
LIN {X 0,Y 474.652,Z 374.86,A -85,B 0,C 180,E1 -7091.678,E2 -7091.678} C_VEL
LIN {X 0,Y 474.696,Z 374.855,A -85,B 0,C 180,E1 -7094.544,E2 -7094.544} C_VEL
LIN {X 0,Y 474.701,Z 374.853,A -85,B 0,C 180,E1 -7098.037,E2 -7098.037} C_VEL
LIN {X 0,Y 474.725,Z 374.853,A -85,B 0,C 180,E1 -7101.486,E2 -7101.486} C_VEL
LIN {X 0,Y 474.778,Z 374.844,A -85,B 0,C 180,E1 -7104.052,E2 -7104.052} C_VEL
LIN {X 0,Y 474.891,Z 374.832,A -85,B 0,C 180,E1 -7107.455,E2 -7107.455} C_VEL
LIN {X 0,Y 474.909,Z 374.828,A -85,B 0,C 180,E1 -7110,E2 -7110} C_VEL
LIN {X 0,Y 474.891,Z 374.832,A -85,B 0,C 180,E1 -7112.544,E2 -7112.544} C_VEL
LIN {X 0,Y 474.778,Z 374.844,A -85,B 0,C 180,E1 -7115.947,E2 -7115.947} C_VEL
LIN {X 0,Y 474.724,Z 374.853,A -85,B 0,C 180,E1 -7118.513,E2 -7118.513} C_VEL
LIN {X 0,Y 474.7,Z 374.853,A -85,B 0,C 180,E1 -7121.962,E2 -7121.962} C_VEL
LIN {X 0,Y 474.695,Z 374.855,A -85,B 0,C 180,E1 -7125.455,E2 -7125.455} C_VEL
LIN {X 0,Y 474.661,Z 374.863,A -85,B 0,C 180,E1 -7129.01,E2 -7129.01} C_VEL
LIN {X 0,Y 474.585,Z 374.867,A -85,B 0,C 180,E1 -7131.729,E2 -7131.729} C_VEL
LIN {X 0,Y 474.654,Z 374.862,A -85,B 0,C 180,E1 -7134.493,E2 -7134.493} C_VEL
LIN {X 0,Y 474.693,Z 374.854,A -85,B 0,C 180,E1 -7137.338,E2 -7137.338} C_VEL
LIN {X 0,Y 474.605,Z 374.865,A -85,B 0,C 180,E1 -7140.811,E2 -7140.811} C_VEL
LIN {X 0,Y 474.632,Z 374.853,A -85,B 0,C 180,E1 -7143.984,E2 -7143.984} C_VEL
LIN {X 0,Y 474.57,Z 374.872,A -85,B 0,C 180,E1 -7146.9,E2 -7146.9} C_VEL
LIN {X 0,Y 474.644,Z 374.854,A -85,B 0,C 180,E1 -7149.651,E2 -7149.651} C_VEL
LIN {X 0,Y 474.6,Z 374.85,A -85,B 0,C 180,E1 -7152.935,E2 -7152.935} C_VEL
LIN {X 0,Y 474.608,Z 374.861,A -85,B 0,C 180,E1 -7155.896,E2 -7155.896} C_VEL
LIN {X 0,Y 474.625,Z 374.857,A -85,B 0,C 180,E1 -7159.04,E2 -7159.04} C_VEL
LIN {X 0,Y 474.604,Z 374.863,A -85,B 0,C 180,E1 -7161.704,E2 -7161.704} C_VEL
LIN {X 0,Y 474.623,Z 374.857,A -85,B 0,C 180,E1 -7164.726,E2 -7164.726} C_VEL
LIN {X 0,Y 474.63,Z 374.858,A -85,B 0,C 180,E1 -7167.788,E2 -7167.788} C_VEL
LIN {X 0,Y 474.625,Z 374.857,A -85,B 0,C 180,E1 -7170.883,E2 -7170.883} C_VEL
LIN {X 0,Y 474.659,Z 374.848,A -85,B 0,C 180,E1 -7173.629,E2 -7173.629} C_VEL
LIN {X 0,Y 474.628,Z 374.865,A -85,B 0,C 180,E1 -7176.641,E2 -7176.641} C_VEL
LIN {X 0,Y 474.65,Z 374.852,A -85,B 0,C 180,E1 -7180.09,E2 -7180.09} C_VEL
LIN {X 0,Y 474.644,Z 374.859,A -85,B 0,C 180,E1 -7182.775,E2 -7182.775} C_VEL
LIN {X 0,Y 474.641,Z 374.857,A -85,B 0,C 180,E1 -7185.421,E2 -7185.421} C_VEL
LIN {X 0,Y 474.732,Z 374.846,A -85,B 0,C 180,E1 -7188.039,E2 -7188.039} C_VEL
LIN {X 0,Y 474.721,Z 374.839,A -85,B 0,C 180,E1 -7191.487,E2 -7191.487} C_VEL
LIN {X 0,Y 474.773,Z 374.843,A -85,B 0,C 180,E1 -7194.053,E2 -7194.053} C_VEL
LIN {X 0,Y 474.889,Z 374.821,A -85,B 0,C 180,E1 -7197.456,E2 -7197.456} C_VEL
LIN {X 0,Y 474.905,Z 374.812,A -85,B 0,C 180,E1 -7200,E2 -7200} C_VEL
LIN {X 0,Y 474.889,Z 374.831,A -85,B 0,C 180,E1 -7202.545,E2 -7202.545} C_VEL
LIN {X 0,Y 474.774,Z 374.844,A -85,B 0,C 180,E1 -7205.948,E2 -7205.948} C_VEL
LIN {X 0,Y 474.722,Z 374.836,A -85,B 0,C 180,E1 -7208.514,E2 -7208.514} C_VEL
LIN {X 0,Y 474.698,Z 374.847,A -85,B 0,C 180,E1 -7211.963,E2 -7211.963} C_VEL
LIN {X 0,Y 474.696,Z 374.851,A -85,B 0,C 180,E1 -7215.778,E2 -7215.778} C_VEL
LIN {X 0,Y 474.661,Z 374.844,A -85,B 0,C 180,E1 -7219.011,E2 -7219.011} C_VEL
LIN {X 0,Y 474.586,Z 374.864,A -85,B 0,C 180,E1 -7221.729,E2 -7221.729} C_VEL
LIN {X 0,Y 474.655,Z 374.854,A -85,B 0,C 180,E1 -7224.494,E2 -7224.494} C_VEL
LIN {X 0,Y 474.695,Z 374.841,A -85,B 0,C 180,E1 -7227.339,E2 -7227.339} C_VEL
LIN {X 0,Y 474.607,Z 374.862,A -85,B 0,C 180,E1 -7230.812,E2 -7230.812} C_VEL
LIN {X 0,Y 474.635,Z 374.855,A -85,B 0,C 180,E1 -7233.985,E2 -7233.985} C_VEL
LIN {X 0,Y 474.572,Z 374.867,A -85,B 0,C 180,E1 -7236.901,E2 -7236.901} C_VEL
LIN {X 0,Y 474.648,Z 374.856,A -85,B 0,C 180,E1 -7239.652,E2 -7239.652} C_VEL
LIN {X 0,Y 474.65,Z 374.856,A -85,B 0,C 180,E1 -7242.931,E2 -7242.931} C_VEL
LIN {X 0,Y 474.608,Z 374.868,A -85,B 0,C 180,E1 -7245.896,E2 -7245.896} C_VEL
LIN {X 0,Y 474.627,Z 374.849,A -85,B 0,C 180,E1 -7249.042,E2 -7249.042} C_VEL
LIN {X 0,Y 474.61,Z 374.866,A -85,B 0,C 180,E1 -7251.705,E2 -7251.705} C_VEL
LIN {X 0,Y 474.63,Z 374.859,A -85,B 0,C 180,E1 -7254.727,E2 -7254.727} C_VEL
LIN {X 0,Y 474.637,Z 374.86,A -85,B 0,C 180,E1 -7257.789,E2 -7257.789} C_VEL
LIN {X 0,Y 474.634,Z 374.864,A -85,B 0,C 180,E1 -7260.883,E2 -7260.883} C_VEL
LIN {X 0,Y 474.716,Z 375.061,A -85,B 0,C 180,E1 -7262.682,E2 -7262.682} C_VEL
LIN {X 0,Y 476.384,Z 384.252,A -85,B 0,C 180,E1 -7264.904,E2 -7264.904} C_VEL
LIN {X 0,Y 476.109,Z 393.528,A -85,B 0,C 180,E1 -7266.973,E2 -7266.973} C_VEL
LIN {X 0,Y 475.54,Z 406.981,A -85,B 0,C 180,E1 -7269.903,E2 -7269.903} C_VEL
LIN {X 0,Y 475.006,Z 420.292,A -85,B 0,C 180,E1 -7272.788,E2 -7272.788} C_VEL
LIN {X 0,Y 474.995,Z 422.438,A -85,B 0,C 180,E1 -7273.22,E2 -7273.22} C_VEL
LIN {X 0,Y 477.034,Z 434.608,A -85,B 0,C 180,E1 -7273.511,E2 -7273.511} C_VEL
LIN {X 0,Y 478.06,Z 441.176,A -85,B 0,C 180,E1 -7273.648,E2 -7273.648} C_VEL
LIN {X 0,Y 477.448,Z 527.248,A -85,B 0,C 180,E1 -7274.964,E2 -7274.964} C_VEL
LIN {X 0,Y 477.224,Z 537.162,A -85,B 0,C 180,E1 -7275.202,E2 -7275.202} C_VEL
LIN {X 0,Y 476.898,Z 547.148,A -85,B 0,C 180,E1 -7275.546,E2 -7275.546} C_VEL
LIN {X 0,Y 476.544,Z 557.507,A -85,B 0,C 180,E1 -7276.026,E2 -7276.026} C_VEL
LIN {X 0,Y 476.151,Z 566.657,A -85,B 0,C 180,E1 -7276.558,E2 -7276.558} C_VEL
LIN {X 0,Y 475.765,Z 575.658,A -85,B 0,C 180,E1 -7277.199,E2 -7277.199} C_VEL
LIN {X 0,Y 475.444,Z 584.475,A -85,B 0,C 180,E1 -7277.957,E2 -7277.957} C_VEL
LIN {X 0,Y 475.152,Z 591.815,A -85,B 0,C 180,E1 -7278.698,E2 -7278.698} C_VEL
LIN {X 0,Y 474.654,Z 600.611,A -85,B 0,C 180,E1 -7279.766,E2 -7279.766} C_VEL
LIN {X 0,Y 474.416,Z 606.603,A -85,B 0,C 180,E1 -7280.622,E2 -7280.622} C_VEL
LIN {X 0,Y 474.175,Z 612.914,A -85,B 0,C 180,E1 -7281.691,E2 -7281.691} C_VEL
LIN {X 0,Y 474.012,Z 618.187,A -85,B 0,C 180,E1 -7282.76,E2 -7282.76} C_VEL
LIN {X 0,Y 473.848,Z 623.278,A -85,B 0,C 180,E1 -7284.041,E2 -7284.041} C_VEL
LIN {X 0,Y 473.763,Z 627.238,A -85,B 0,C 180,E1 -7285.32,E2 -7285.32} C_VEL
LIN {X 0,Y 473.795,Z 630.169,A -85,B 0,C 180,E1 -7286.599,E2 -7286.599} C_VEL
LIN {X 0,Y 473.741,Z 631.665,A -85,B 0,C 180,E1 -7287.449,E2 -7287.449} C_VEL
LIN {X 0,Y 473.688,Z 633.182,A -85,B 0,C 180,E1 -7289.15,E2 -7289.15} C_VEL
LIN {X 0,Y 473.669,Z 633.46,A -85,B 0,C 180,E1 -7290,E2 -7290} C_VEL
LIN {X 0,Y 473.698,Z 632.589,A -85,B 0,C 180,E1 -7291.701,E2 -7291.701} C_VEL
LIN {X 0,Y 473.741,Z 631.664,A -85,B 0,C 180,E1 -7292.551,E2 -7292.551} C_VEL
LIN {X 0,Y 473.796,Z 630.168,A -85,B 0,C 180,E1 -7293.402,E2 -7293.402} C_VEL
LIN {X 0,Y 473.83,Z 626.115,A -85,B 0,C 180,E1 -7295.106,E2 -7295.106} C_VEL
LIN {X 0,Y 473.881,Z 621.484,A -85,B 0,C 180,E1 -7296.453,E2 -7296.453} C_VEL
LIN {X 0,Y 474.052,Z 616.188,A -85,B 0,C 180,E1 -7297.668,E2 -7297.668} C_VEL
LIN {X 0,Y 474.284,Z 610.536,A -85,B 0,C 180,E1 -7298.736,E2 -7298.736} C_VEL
LIN {X 0,Y 474.55,Z 603.73,A -85,B 0,C 180,E1 -7299.806,E2 -7299.806} C_VEL
LIN {X 0,Y 474.9,Z 595.51,A -85,B 0,C 180,E1 -7300.876,E2 -7300.876} C_VEL
LIN {X 0,Y 475.304,Z 587.682,A -85,B 0,C 180,E1 -7301.731,E2 -7301.731} C_VEL
LIN {X 0,Y 475.672,Z 579.728,A -85,B 0,C 180,E1 -7302.468,E2 -7302.468} C_VEL
LIN {X 0,Y 476.076,Z 569.835,A -85,B 0,C 180,E1 -7303.227,E2 -7303.227} C_VEL
LIN {X 0,Y 476.389,Z 561.435,A -85,B 0,C 180,E1 -7303.762,E2 -7303.762} C_VEL
LIN {X 0,Y 476.82,Z 550.926,A -85,B 0,C 180,E1 -7304.293,E2 -7304.293} C_VEL
LIN {X 0,Y 477.099,Z 540.589,A -85,B 0,C 180,E1 -7304.693,E2 -7304.693} C_VEL
LIN {X 0,Y 477.418,Z 529.867,A -85,B 0,C 180,E1 -7304.983,E2 -7304.983} C_VEL
LIN {X 0,Y 477.634,Z 505.624,A -85,B 0,C 180,E1 -7305.381,E2 -7305.381} C_VEL
LIN {X 0,Y 477.955,Z 440.238,A -85,B 0,C 180,E1 -7306.37,E2 -7306.37} C_VEL
LIN {X 0,Y 474.999,Z 422.598,A -85,B 0,C 180,E1 -7306.767,E2 -7306.767} C_VEL
LIN {X 0,Y 474.974,Z 421.736,A -85,B 0,C 180,E1 -7306.881,E2 -7306.881} C_VEL
LIN {X 0,Y 475.483,Z 409.19,A -85,B 0,C 180,E1 -7309.649,E2 -7309.649} C_VEL
LIN {X 0,Y 476.068,Z 394.596,A -85,B 0,C 180,E1 -7312.8,E2 -7312.8} C_VEL
LIN {X 0,Y 476.434,Z 385.272,A -85,B 0,C 180,E1 -7314.86,E2 -7314.86} C_VEL
LIN {X 0,Y 475.284,Z 378.093,A -85,B 0,C 180,E1 -7316.571,E2 -7316.571} C_VEL
LIN {X 0,Y 474.698,Z 374.965,A -85,B 0,C 180,E1 -7317.368,E2 -7317.368} C_VEL
LIN {X 0,Y 474.616,Z 374.864,A -85,B 0,C 180,E1 -7320.229,E2 -7320.229} C_VEL
LIN {X 0,Y 474.645,Z 374.856,A -85,B 0,C 180,E1 -7323.22,E2 -7323.22} C_VEL
LIN {X 0,Y 474.596,Z 374.863,A -85,B 0,C 180,E1 -7326.323,E2 -7326.323} C_VEL
LIN {X 0,Y 474.63,Z 374.86,A -85,B 0,C 180,E1 -7329.647,E2 -7329.647} C_VEL
LIN {X 0,Y 474.616,Z 374.86,A -85,B 0,C 180,E1 -7332.934,E2 -7332.934} C_VEL
LIN {X 0,Y 474.619,Z 374.863,A -85,B 0,C 180,E1 -7335.896,E2 -7335.896} C_VEL
LIN {X 0,Y 474.647,Z 374.856,A -85,B 0,C 180,E1 -7339.038,E2 -7339.038} C_VEL
LIN {X 0,Y 474.617,Z 374.862,A -85,B 0,C 180,E1 -7341.703,E2 -7341.703} C_VEL
LIN {X 0,Y 474.629,Z 374.855,A -85,B 0,C 180,E1 -7344.726,E2 -7344.726} C_VEL
LIN {X 0,Y 474.638,Z 374.859,A -85,B 0,C 180,E1 -7347.787,E2 -7347.787} C_VEL
LIN {X 0,Y 474.632,Z 374.857,A -85,B 0,C 180,E1 -7350.882,E2 -7350.882} C_VEL
LIN {X 0,Y 474.66,Z 374.848,A -85,B 0,C 180,E1 -7353.628,E2 -7353.628} C_VEL
LIN {X 0,Y 474.635,Z 374.857,A -85,B 0,C 180,E1 -7356.641,E2 -7356.641} C_VEL
LIN {X 0,Y 474.654,Z 374.849,A -85,B 0,C 180,E1 -7360.089,E2 -7360.089} C_VEL
LIN {X 0,Y 474.649,Z 374.847,A -85,B 0,C 180,E1 -7362.774,E2 -7362.774} C_VEL
LIN {X 0,Y 474.647,Z 374.858,A -85,B 0,C 180,E1 -7365.42,E2 -7365.42} C_VEL
LIN {X 0,Y 474.702,Z 374.847,A -85,B 0,C 180,E1 -7368.037,E2 -7368.037} C_VEL
LIN {X 0,Y 474.726,Z 374.834,A -85,B 0,C 180,E1 -7371.486,E2 -7371.486} C_VEL
LIN {X 0,Y 474.777,Z 374.844,A -85,B 0,C 180,E1 -7374.052,E2 -7374.052} C_VEL
LIN {X 0,Y 474.892,Z 374.831,A -85,B 0,C 180,E1 -7377.455,E2 -7377.455} C_VEL
LIN {X 0,Y 474.909,Z 374.811,A -85,B 0,C 180,E1 -7380,E2 -7380} C_VEL
LIN {X 0,Y 474.892,Z 374.821,A -85,B 0,C 180,E1 -7382.544,E2 -7382.544} C_VEL
LIN {X 0,Y 474.776,Z 374.843,A -85,B 0,C 180,E1 -7385.947,E2 -7385.947} C_VEL
LIN {X 0,Y 474.725,Z 374.839,A -85,B 0,C 180,E1 -7388.513,E2 -7388.513} C_VEL
LIN {X 0,Y 474.736,Z 374.845,A -85,B 0,C 180,E1 -7391.961,E2 -7391.961} C_VEL
LIN {X 0,Y 474.677,Z 374.856,A -85,B 0,C 180,E1 -7395.768,E2 -7395.768} C_VEL
LIN {X 0,Y 474.661,Z 374.846,A -85,B 0,C 180,E1 -7399.01,E2 -7399.01} C_VEL
LIN {X 0,Y 474.586,Z 374.869,A -85,B 0,C 180,E1 -7401.728,E2 -7401.728} C_VEL
LIN {X 0,Y 474.655,Z 374.855,A -85,B 0,C 180,E1 -7404.492,E2 -7404.492} C_VEL
LIN {X 0,Y 474.695,Z 374.846,A -85,B 0,C 180,E1 -7407.338,E2 -7407.338} C_VEL
LIN {X 0,Y 474.601,Z 374.864,A -85,B 0,C 180,E1 -7410.81,E2 -7410.81} C_VEL
LIN {X 0,Y 474.634,Z 374.851,A -85,B 0,C 180,E1 -7413.984,E2 -7413.984} C_VEL
LIN {X 0,Y 474.571,Z 374.867,A -85,B 0,C 180,E1 -7416.9,E2 -7416.9} C_VEL
LIN {X 0,Y 474.623,Z 374.858,A -85,B 0,C 180,E1 -7419.647,E2 -7419.647} C_VEL
LIN {X 0,Y 474.631,Z 374.861,A -85,B 0,C 180,E1 -7422.932,E2 -7422.932} C_VEL
LIN {X 0,Y 474.604,Z 374.854,A -85,B 0,C 180,E1 -7425.895,E2 -7425.895} C_VEL
LIN {X 0,Y 474.637,Z 374.843,A -85,B 0,C 180,E1 -7429.039,E2 -7429.039} C_VEL
LIN {X 0,Y 474.613,Z 374.865,A -85,B 0,C 180,E1 -7431.703,E2 -7431.703} C_VEL
LIN {X 0,Y 474.626,Z 374.855,A -85,B 0,C 180,E1 -7434.726,E2 -7434.726} C_VEL
LIN {X 0,Y 474.634,Z 374.862,A -85,B 0,C 180,E1 -7437.788,E2 -7437.788} C_VEL
LIN {X 0,Y 474.628,Z 374.854,A -85,B 0,C 180,E1 -7440.883,E2 -7440.883} C_VEL
LIN {X 0,Y 474.657,Z 374.86,A -85,B 0,C 180,E1 -7443.628,E2 -7443.628} C_VEL
LIN {X 0,Y 474.632,Z 374.863,A -85,B 0,C 180,E1 -7446.641,E2 -7446.641} C_VEL
LIN {X 0,Y 474.653,Z 374.859,A -85,B 0,C 180,E1 -7450.09,E2 -7450.09} C_VEL
LIN {X 0,Y 474.652,Z 374.86,A -85,B 0,C 180,E1 -7451.678,E2 -7451.678} C_VEL
LIN {X 0,Y 473.99,Z 374.943,A -85,B 0,C 180,E1 -7452.387,E2 -7452.387} C_VEL
LIN {X 0,Y 471.139,Z 375.3,A -85,B 0,C 180,E1 -7453.539,E2 -7453.539} C_VEL
LIN {X 0,Y 468.722,Z 375.604,A -85,B 0,C 180,E1 -7454.467,E2 -7454.467} C_VEL
LIN {X 0,Y 467.68,Z 375.732,A -85,B 0,C 180,E1 -7455.184,E2 -7455.184} C_VEL
LIN {X 0,Y 467.593,Z 375.74,A -85,B 0,C 180,E1 -7455.427,E2 -7455.427} C_VEL
LIN {X 0,Y 467.65,Z 375.735,A -85,B 0,C 180,E1 -7458.734,E2 -7458.734} C_VEL
LIN {X 0,Y 467.745,Z 375.721,A -85,B 0,C 180,E1 -7462.228,E2 -7462.228} C_VEL
LIN {X 0,Y 467.723,Z 375.726,A -85,B 0,C 180,E1 -7464.827,E2 -7464.827} C_VEL
LIN {X 0,Y 467.857,Z 375.709,A -85,B 0,C 180,E1 -7467.417,E2 -7467.417} C_VEL
LIN {X 0,Y 467.88,Z 375.704,A -85,B 0,C 180,E1 -7470,E2 -7470} C_VEL
LIN {X 0,Y 467.857,Z 375.709,A -85,B 0,C 180,E1 -7472.583,E2 -7472.583} C_VEL
LIN {X 0,Y 467.742,Z 375.72,A -85,B 0,C 180,E1 -7476.037,E2 -7476.037} C_VEL
LIN {X 0,Y 467.678,Z 375.732,A -85,B 0,C 180,E1 -7478.642,E2 -7478.642} C_VEL
LIN {X 0,Y 467.652,Z 375.732,A -85,B 0,C 180,E1 -7482.145,E2 -7482.145} C_VEL
LIN {X 0,Y 467.635,Z 375.733,A -85,B 0,C 180,E1 -7485.695,E2 -7485.695} C_VEL
LIN {X 0,Y 467.613,Z 375.74,A -85,B 0,C 180,E1 -7488.765,E2 -7488.765} C_VEL
LIN {X 0,Y 467.576,Z 375.743,A -85,B 0,C 180,E1 -7491.268,E2 -7491.268} C_VEL
LIN {X 0,Y 467.568,Z 375.741,A -85,B 0,C 180,E1 -7493.943,E2 -7493.943} C_VEL
LIN {X 0,Y 467.623,Z 375.739,A -85,B 0,C 180,E1 -7496.799,E2 -7496.799} C_VEL
LIN {X 0,Y 467.582,Z 375.73,A -85,B 0,C 180,E1 -7499.735,E2 -7499.735} C_VEL
LIN {X 0,Y 467.578,Z 375.74,A -85,B 0,C 180,E1 -7502.758,E2 -7502.758} C_VEL
LIN {X 0,Y 467.55,Z 375.735,A -85,B 0,C 180,E1 -7505.889,E2 -7505.889} C_VEL
LIN {X 0,Y 467.609,Z 375.733,A -85,B 0,C 180,E1 -7509.141,E2 -7509.141} C_VEL
LIN {X 0,Y 467.579,Z 375.719,A -85,B 0,C 180,E1 -7512.567,E2 -7512.567} C_VEL
LIN {X 0,Y 467.564,Z 375.742,A -85,B 0,C 180,E1 -7515.053,E2 -7515.053} C_VEL
LIN {X 0,Y 467.581,Z 375.736,A -85,B 0,C 180,E1 -7517.44,E2 -7517.44} C_VEL
LIN {X 0,Y 467.585,Z 375.742,A -85,B 0,C 180,E1 -7520.856,E2 -7520.856} C_VEL
LIN {X 0,Y 467.556,Z 375.743,A -85,B 0,C 180,E1 -7524.26,E2 -7524.26} C_VEL
LIN {X 0,Y 467.575,Z 375.738,A -85,B 0,C 180,E1 -7527.321,E2 -7527.321} C_VEL
LIN {X 0,Y 467.571,Z 375.739,A -85,B 0,C 180,E1 -7530.666,E2 -7530.666} C_VEL
LIN {X 0,Y 467.62,Z 375.726,A -85,B 0,C 180,E1 -7533.201,E2 -7533.201} C_VEL
LIN {X 0,Y 467.585,Z 375.744,A -85,B 0,C 180,E1 -7536.468,E2 -7536.468} C_VEL
LIN {X 0,Y 467.617,Z 375.725,A -85,B 0,C 180,E1 -7539.777,E2 -7539.777} C_VEL
LIN {X 0,Y 467.602,Z 375.732,A -85,B 0,C 180,E1 -7542.507,E2 -7542.507} C_VEL
LIN {X 0,Y 467.599,Z 375.735,A -85,B 0,C 180,E1 -7545.197,E2 -7545.197} C_VEL
LIN {X 0,Y 467.676,Z 375.723,A -85,B 0,C 180,E1 -7547.856,E2 -7547.856} C_VEL
LIN {X 0,Y 467.675,Z 375.717,A -85,B 0,C 180,E1 -7551.358,E2 -7551.358} C_VEL
LIN {X 0,Y 467.737,Z 375.719,A -85,B 0,C 180,E1 -7553.963,E2 -7553.963} C_VEL
LIN {X 0,Y 467.855,Z 375.697,A -85,B 0,C 180,E1 -7557.418,E2 -7557.418} C_VEL
LIN {X 0,Y 467.876,Z 375.686,A -85,B 0,C 180,E1 -7560,E2 -7560} C_VEL
LIN {X 0,Y 467.855,Z 375.707,A -85,B 0,C 180,E1 -7562.583,E2 -7562.583} C_VEL
LIN {X 0,Y 467.738,Z 375.721,A -85,B 0,C 180,E1 -7566.038,E2 -7566.038} C_VEL
LIN {X 0,Y 467.676,Z 375.711,A -85,B 0,C 180,E1 -7568.643,E2 -7568.643} C_VEL
LIN {X 0,Y 467.65,Z 375.728,A -85,B 0,C 180,E1 -7572.146,E2 -7572.146} C_VEL
LIN {X 0,Y 467.662,Z 375.728,A -85,B 0,C 180,E1 -7575.893,E2 -7575.893} C_VEL
LIN {X 0,Y 467.619,Z 375.72,A -85,B 0,C 180,E1 -7579.308,E2 -7579.308} C_VEL
LIN {X 0,Y 467.533,Z 375.747,A -85,B 0,C 180,E1 -7582.074,E2 -7582.074} C_VEL
LIN {X 0,Y 467.599,Z 375.73,A -85,B 0,C 180,E1 -7584.888,E2 -7584.888} C_VEL
LIN {X 0,Y 467.625,Z 375.724,A -85,B 0,C 180,E1 -7587.769,E2 -7587.769} C_VEL
LIN {X 0,Y 467.569,Z 375.738,A -85,B 0,C 180,E1 -7591.047,E2 -7591.047} C_VEL
LIN {X 0,Y 467.587,Z 375.734,A -85,B 0,C 180,E1 -7594.243,E2 -7594.243} C_VEL
LIN {X 0,Y 467.548,Z 375.741,A -85,B 0,C 180,E1 -7597.188,E2 -7597.188} C_VEL
LIN {X 0,Y 467.594,Z 375.737,A -85,B 0,C 180,E1 -7600.263,E2 -7600.263} C_VEL
LIN {X 0,Y 467.617,Z 375.734,A -85,B 0,C 180,E1 -7602.572,E2 -7602.572} C_VEL
LIN {X 0,Y 467.569,Z 375.738,A -85,B 0,C 180,E1 -7605.054,E2 -7605.054} C_VEL
LIN {X 0,Y 467.587,Z 375.738,A -85,B 0,C 180,E1 -7607.441,E2 -7607.441} C_VEL
LIN {X 0,Y 467.582,Z 375.737,A -85,B 0,C 180,E1 -7610.856,E2 -7610.856} C_VEL
LIN {X 0,Y 467.563,Z 375.738,A -85,B 0,C 180,E1 -7614.261,E2 -7614.261} C_VEL
LIN {X 0,Y 467.582,Z 375.736,A -85,B 0,C 180,E1 -7617.322,E2 -7617.322} C_VEL
LIN {X 0,Y 467.58,Z 375.743,A -85,B 0,C 180,E1 -7620.666,E2 -7620.666} C_VEL
LIN {X 0,Y 467.681,Z 375.877,A -85,B 0,C 180,E1 -7622.451,E2 -7622.451} C_VEL
LIN {X 0,Y 469.369,Z 385.133,A -85,B 0,C 180,E1 -7624.74,E2 -7624.74} C_VEL
LIN {X 0,Y 469.249,Z 392.319,A -85,B 0,C 180,E1 -7626.383,E2 -7626.383} C_VEL
LIN {X 0,Y 468.602,Z 406.811,A -85,B 0,C 180,E1 -7629.593,E2 -7629.593} C_VEL
LIN {X 0,Y 468.026,Z 420.102,A -85,B 0,C 180,E1 -7632.523,E2 -7632.523} C_VEL
LIN {X 0,Y 467.944,Z 422.089,A -85,B 0,C 180,E1 -7632.942,E2 -7632.942} C_VEL
LIN {X 0,Y 468.592,Z 425.821,A -85,B 0,C 180,E1 -7633.072,E2 -7633.072} C_VEL
LIN {X 0,Y 471.24,Z 442.063,A -85,B 0,C 180,E1 -7633.421,E2 -7633.421} C_VEL
LIN {X 0,Y 470.59,Z 527.053,A -85,B 0,C 180,E1 -7634.739,E2 -7634.739} C_VEL
LIN {X 0,Y 470.375,Z 536.967,A -85,B 0,C 180,E1 -7634.982,E2 -7634.982} C_VEL
LIN {X 0,Y 470.006,Z 546.953,A -85,B 0,C 180,E1 -7635.33,E2 -7635.33} C_VEL
LIN {X 0,Y 469.641,Z 557.311,A -85,B 0,C 180,E1 -7635.816,E2 -7635.816} C_VEL
LIN {X 0,Y 469.219,Z 566.458,A -85,B 0,C 180,E1 -7636.355,E2 -7636.355} C_VEL
LIN {X 0,Y 468.828,Z 575.463,A -85,B 0,C 180,E1 -7637.006,E2 -7637.006} C_VEL
LIN {X 0,Y 468.535,Z 583.482,A -85,B 0,C 180,E1 -7637.697,E2 -7637.697} C_VEL
LIN {X 0,Y 468.154,Z 591.619,A -85,B 0,C 180,E1 -7638.527,E2 -7638.527} C_VEL
LIN {X 0,Y 467.63,Z 600.415,A -85,B 0,C 180,E1 -7639.61,E2 -7639.61} C_VEL
LIN {X 0,Y 467.382,Z 606.407,A -85,B 0,C 180,E1 -7640.48,E2 -7640.48} C_VEL
LIN {X 0,Y 467.12,Z 612.718,A -85,B 0,C 180,E1 -7641.565,E2 -7641.565} C_VEL
LIN {X 0,Y 466.94,Z 617.991,A -85,B 0,C 180,E1 -7642.65,E2 -7642.65} C_VEL
LIN {X 0,Y 466.764,Z 623.082,A -85,B 0,C 180,E1 -7643.95,E2 -7643.95} C_VEL
LIN {X 0,Y 466.691,Z 627.043,A -85,B 0,C 180,E1 -7645.249,E2 -7645.249} C_VEL
LIN {X 0,Y 466.689,Z 629.974,A -85,B 0,C 180,E1 -7646.547,E2 -7646.547} C_VEL
LIN {X 0,Y 466.662,Z 631.47,A -85,B 0,C 180,E1 -7647.411,E2 -7647.411} C_VEL
LIN {X 0,Y 466.619,Z 632.988,A -85,B 0,C 180,E1 -7649.137,E2 -7649.137} C_VEL
LIN {X 0,Y 466.598,Z 633.266,A -85,B 0,C 180,E1 -7650,E2 -7650} C_VEL
LIN {X 0,Y 466.607,Z 632.394,A -85,B 0,C 180,E1 -7651.726,E2 -7651.726} C_VEL
LIN {X 0,Y 466.662,Z 631.47,A -85,B 0,C 180,E1 -7652.59,E2 -7652.59} C_VEL
LIN {X 0,Y 466.647,Z 628.128,A -85,B 0,C 180,E1 -7654.319,E2 -7654.319} C_VEL
LIN {X 0,Y 466.769,Z 624.508,A -85,B 0,C 180,E1 -7655.617,E2 -7655.617} C_VEL
LIN {X 0,Y 466.806,Z 621.697,A -85,B 0,C 180,E1 -7656.451,E2 -7656.451} C_VEL
LIN {X 0,Y 466.995,Z 615.992,A -85,B 0,C 180,E1 -7657.784,E2 -7657.784} C_VEL
LIN {X 0,Y 467.224,Z 610.34,A -85,B 0,C 180,E1 -7658.869,E2 -7658.869} C_VEL
LIN {X 0,Y 467.527,Z 603.534,A -85,B 0,C 180,E1 -7659.955,E2 -7659.955} C_VEL
LIN {X 0,Y 467.907,Z 595.315,A -85,B 0,C 180,E1 -7661.041,E2 -7661.041} C_VEL
LIN {X 0,Y 468.325,Z 587.486,A -85,B 0,C 180,E1 -7661.908,E2 -7661.908} C_VEL
LIN {X 0,Y 468.697,Z 579.569,A -85,B 0,C 180,E1 -7662.654,E2 -7662.654} C_VEL
LIN {X 0,Y 469.144,Z 569.64,A -85,B 0,C 180,E1 -7663.426,E2 -7663.426} C_VEL
LIN {X 0,Y 469.478,Z 561.239,A -85,B 0,C 180,E1 -7663.969,E2 -7663.969} C_VEL
LIN {X 0,Y 469.922,Z 550.73,A -85,B 0,C 180,E1 -7664.508,E2 -7664.508} C_VEL
LIN {X 0,Y 470.233,Z 540.394,A -85,B 0,C 180,E1 -7664.913,E2 -7664.913} C_VEL
LIN {X 0,Y 470.559,Z 529.671,A -85,B 0,C 180,E1 -7665.207,E2 -7665.207} C_VEL
LIN {X 0,Y 470.795,Z 505.512,A -85,B 0,C 180,E1 -7665.609,E2 -7665.609} C_VEL
LIN {X 0,Y 471.094,Z 440.751,A -85,B 0,C 180,E1 -7666.604,E2 -7666.604} C_VEL
LIN {X 0,Y 468.011,Z 422.472,A -85,B 0,C 180,E1 -7667.021,E2 -7667.021} C_VEL
LIN {X 0,Y 467.985,Z 420.964,A -85,B 0,C 180,E1 -7667.276,E2 -7667.276} C_VEL
LIN {X 0,Y 468.465,Z 410.055,A -85,B 0,C 180,E1 -7669.728,E2 -7669.728} C_VEL
LIN {X 0,Y 469.121,Z 395.507,A -85,B 0,C 180,E1 -7672.924,E2 -7672.924} C_VEL
LIN {X 0,Y 469.463,Z 386.154,A -85,B 0,C 180,E1 -7675.018,E2 -7675.018} C_VEL
LIN {X 0,Y 468.248,Z 378.973,A -85,B 0,C 180,E1 -7676.761,E2 -7676.761} C_VEL
LIN {X 0,Y 467.652,Z 375.823,A -85,B 0,C 180,E1 -7677.611,E2 -7677.611} C_VEL
LIN {X 0,Y 467.575,Z 375.742,A -85,B 0,C 180,E1 -7681.045,E2 -7681.045} C_VEL
LIN {X 0,Y 467.593,Z 375.741,A -85,B 0,C 180,E1 -7684.242,E2 -7684.242} C_VEL
LIN {X 0,Y 467.553,Z 375.74,A -85,B 0,C 180,E1 -7687.186,E2 -7687.186} C_VEL
LIN {X 0,Y 467.579,Z 375.729,A -85,B 0,C 180,E1 -7690.264,E2 -7690.264} C_VEL
LIN {X 0,Y 467.588,Z 375.737,A -85,B 0,C 180,E1 -7692.567,E2 -7692.567} C_VEL
LIN {X 0,Y 467.572,Z 375.737,A -85,B 0,C 180,E1 -7695.053,E2 -7695.053} C_VEL
LIN {X 0,Y 467.626,Z 375.733,A -85,B 0,C 180,E1 -7697.444,E2 -7697.444} C_VEL
LIN {X 0,Y 467.6,Z 375.731,A -85,B 0,C 180,E1 -7700.857,E2 -7700.857} C_VEL
LIN {X 0,Y 467.563,Z 375.739,A -85,B 0,C 180,E1 -7704.26,E2 -7704.26} C_VEL
LIN {X 0,Y 467.583,Z 375.732,A -85,B 0,C 180,E1 -7707.32,E2 -7707.32} C_VEL
LIN {X 0,Y 467.578,Z 375.736,A -85,B 0,C 180,E1 -7710.665,E2 -7710.665} C_VEL
LIN {X 0,Y 467.616,Z 375.723,A -85,B 0,C 180,E1 -7713.199,E2 -7713.199} C_VEL
LIN {X 0,Y 467.592,Z 375.736,A -85,B 0,C 180,E1 -7716.468,E2 -7716.468} C_VEL
LIN {X 0,Y 467.622,Z 375.729,A -85,B 0,C 180,E1 -7719.777,E2 -7719.777} C_VEL
LIN {X 0,Y 467.608,Z 375.725,A -85,B 0,C 180,E1 -7722.506,E2 -7722.506} C_VEL
LIN {X 0,Y 467.605,Z 375.733,A -85,B 0,C 180,E1 -7725.196,E2 -7725.196} C_VEL
LIN {X 0,Y 467.654,Z 375.727,A -85,B 0,C 180,E1 -7727.854,E2 -7727.854} C_VEL
LIN {X 0,Y 467.68,Z 375.709,A -85,B 0,C 180,E1 -7731.357,E2 -7731.357} C_VEL
LIN {X 0,Y 467.741,Z 375.721,A -85,B 0,C 180,E1 -7733.962,E2 -7733.962} C_VEL
LIN {X 0,Y 467.857,Z 375.706,A -85,B 0,C 180,E1 -7737.417,E2 -7737.417} C_VEL
LIN {X 0,Y 467.879,Z 375.686,A -85,B 0,C 180,E1 -7740,E2 -7740} C_VEL
LIN {X 0,Y 467.858,Z 375.697,A -85,B 0,C 180,E1 -7742.582,E2 -7742.582} C_VEL
LIN {X 0,Y 467.741,Z 375.718,A -85,B 0,C 180,E1 -7746.037,E2 -7746.037} C_VEL
LIN {X 0,Y 467.679,Z 375.716,A -85,B 0,C 180,E1 -7748.642,E2 -7748.642} C_VEL
LIN {X 0,Y 467.68,Z 375.722,A -85,B 0,C 180,E1 -7752.144,E2 -7752.144} C_VEL
LIN {X 0,Y 467.646,Z 375.73,A -85,B 0,C 180,E1 -7755.885,E2 -7755.885} C_VEL
LIN {X 0,Y 467.62,Z 375.723,A -85,B 0,C 180,E1 -7759.307,E2 -7759.307} C_VEL
LIN {X 0,Y 467.531,Z 375.744,A -85,B 0,C 180,E1 -7762.073,E2 -7762.073} C_VEL
LIN {X 0,Y 467.6,Z 375.735,A -85,B 0,C 180,E1 -7764.887,E2 -7764.887} C_VEL
LIN {X 0,Y 467.623,Z 375.727,A -85,B 0,C 180,E1 -7767.768,E2 -7767.768} C_VEL
LIN {X 0,Y 467.565,Z 375.742,A -85,B 0,C 180,E1 -7771.045,E2 -7771.045} C_VEL
LIN {X 0,Y 467.585,Z 375.727,A -85,B 0,C 180,E1 -7774.242,E2 -7774.242} C_VEL
LIN {X 0,Y 467.546,Z 375.746,A -85,B 0,C 180,E1 -7777.186,E2 -7777.186} C_VEL
LIN {X 0,Y 467.574,Z 375.732,A -85,B 0,C 180,E1 -7780.264,E2 -7780.264} C_VEL
LIN {X 0,Y 467.582,Z 375.736,A -85,B 0,C 180,E1 -7782.567,E2 -7782.567} C_VEL
LIN {X 0,Y 467.567,Z 375.743,A -85,B 0,C 180,E1 -7785.053,E2 -7785.053} C_VEL
LIN {X 0,Y 467.584,Z 375.718,A -85,B 0,C 180,E1 -7787.44,E2 -7787.44} C_VEL
LIN {X 0,Y 467.611,Z 375.733,A -85,B 0,C 180,E1 -7790.858,E2 -7790.858} C_VEL
LIN {X 0,Y 467.559,Z 375.733,A -85,B 0,C 180,E1 -7794.26,E2 -7794.26} C_VEL
LIN {X 0,Y 467.578,Z 375.741,A -85,B 0,C 180,E1 -7797.321,E2 -7797.321} C_VEL
LIN {X 0,Y 467.575,Z 375.732,A -85,B 0,C 180,E1 -7800.665,E2 -7800.665} C_VEL
LIN {X 0,Y 467.613,Z 375.741,A -85,B 0,C 180,E1 -7803.2,E2 -7803.2} C_VEL
LIN {X 0,Y 467.589,Z 375.739,A -85,B 0,C 180,E1 -7806.468,E2 -7806.468} C_VEL
LIN {X 0,Y 467.621,Z 375.736,A -85,B 0,C 180,E1 -7809.777,E2 -7809.777} C_VEL
LIN {X 0,Y 467.606,Z 375.738,A -85,B 0,C 180,E1 -7812.507,E2 -7812.507} C_VEL
LIN {X 0,Y 467.593,Z 375.74,A -85,B 0,C 180,E1 -7815.427,E2 -7815.427} C_VEL
LIN {X 0,Y 466.923,Z 375.822,A -85,B 0,C 180,E1 -7816.146,E2 -7816.146} C_VEL
LIN {X 0,Y 464.08,Z 376.18,A -85,B 0,C 180,E1 -7817.315,E2 -7817.315} C_VEL
LIN {X 0,Y 461.681,Z 376.477,A -85,B 0,C 180,E1 -7818.257,E2 -7818.257} C_VEL
LIN {X 0,Y 460.655,Z 376.607,A -85,B 0,C 180,E1 -7818.984,E2 -7818.984} C_VEL
LIN {X 0,Y 460.574,Z 376.615,A -85,B 0,C 180,E1 -7819.231,E2 -7819.231} C_VEL
LIN {X 0,Y 460.716,Z 376.598,A -85,B 0,C 180,E1 -7822.538,E2 -7822.538} C_VEL
LIN {X 0,Y 460.696,Z 376.602,A -85,B 0,C 180,E1 -7824.748,E2 -7824.748} C_VEL
LIN {X 0,Y 460.822,Z 376.586,A -85,B 0,C 180,E1 -7827.377,E2 -7827.377} C_VEL
LIN {X 0,Y 460.85,Z 376.58,A -85,B 0,C 180,E1 -7830,E2 -7830} C_VEL
LIN {X 0,Y 460.822,Z 376.586,A -85,B 0,C 180,E1 -7832.622,E2 -7832.622} C_VEL
LIN {X 0,Y 460.708,Z 376.597,A -85,B 0,C 180,E1 -7836.13,E2 -7836.13} C_VEL
LIN {X 0,Y 460.625,Z 376.611,A -85,B 0,C 180,E1 -7838.776,E2 -7838.776} C_VEL
LIN {X 0,Y 460.609,Z 376.611,A -85,B 0,C 180,E1 -7842.445,E2 -7842.445} C_VEL
LIN {X 0,Y 460.595,Z 376.61,A -85,B 0,C 180,E1 -7845.997,E2 -7845.997} C_VEL
LIN {X 0,Y 460.567,Z 376.618,A -85,B 0,C 180,E1 -7848.902,E2 -7848.902} C_VEL
LIN {X 0,Y 460.511,Z 376.622,A -85,B 0,C 180,E1 -7851.485,E2 -7851.485} C_VEL
LIN {X 0,Y 460.538,Z 376.619,A -85,B 0,C 180,E1 -7854.332,E2 -7854.332} C_VEL
LIN {X 0,Y 460.579,Z 376.613,A -85,B 0,C 180,E1 -7857.243,E2 -7857.243} C_VEL
LIN {X 0,Y 460.522,Z 376.612,A -85,B 0,C 180,E1 -7860.238,E2 -7860.238} C_VEL
LIN {X 0,Y 460.523,Z 376.611,A -85,B 0,C 180,E1 -7863.325,E2 -7863.325} C_VEL
LIN {X 0,Y 460.473,Z 376.621,A -85,B 0,C 180,E1 -7866.529,E2 -7866.529} C_VEL
LIN {X 0,Y 460.569,Z 376.607,A -85,B 0,C 180,E1 -7869.858,E2 -7869.858} C_VEL
LIN {X 0,Y 460.505,Z 376.603,A -85,B 0,C 180,E1 -7872.9,E2 -7872.9} C_VEL
LIN {X 0,Y 460.512,Z 376.617,A -85,B 0,C 180,E1 -7875.829,E2 -7875.829} C_VEL
LIN {X 0,Y 460.527,Z 376.612,A -85,B 0,C 180,E1 -7878.989,E2 -7878.989} C_VEL
LIN {X 0,Y 460.524,Z 376.618,A -85,B 0,C 180,E1 -7881.267,E2 -7881.267} C_VEL
LIN {X 0,Y 460.506,Z 376.617,A -85,B 0,C 180,E1 -7884.555,E2 -7884.555} C_VEL
LIN {X 0,Y 460.525,Z 376.615,A -85,B 0,C 180,E1 -7887.716,E2 -7887.716} C_VEL
LIN {X 0,Y 460.54,Z 376.613,A -85,B 0,C 180,E1 -7890.77,E2 -7890.77} C_VEL
LIN {X 0,Y 460.561,Z 376.604,A -85,B 0,C 180,E1 -7893.735,E2 -7893.735} C_VEL
LIN {X 0,Y 460.539,Z 376.62,A -85,B 0,C 180,E1 -7896.624,E2 -7896.624} C_VEL
LIN {X 0,Y 460.545,Z 376.605,A -85,B 0,C 180,E1 -7899.453,E2 -7899.453} C_VEL
LIN {X 0,Y 460.552,Z 376.606,A -85,B 0,C 180,E1 -7902.23,E2 -7902.23} C_VEL
LIN {X 0,Y 460.558,Z 376.614,A -85,B 0,C 180,E1 -7904.965,E2 -7904.965} C_VEL
LIN {X 0,Y 460.622,Z 376.6,A -85,B 0,C 180,E1 -7907.667,E2 -7907.667} C_VEL
LIN {X 0,Y 460.622,Z 376.595,A -85,B 0,C 180,E1 -7911.224,E2 -7911.224} C_VEL
LIN {X 0,Y 460.703,Z 376.594,A -85,B 0,C 180,E1 -7913.871,E2 -7913.871} C_VEL
LIN {X 0,Y 460.82,Z 376.573,A -85,B 0,C 180,E1 -7917.378,E2 -7917.378} C_VEL
LIN {X 0,Y 460.847,Z 376.561,A -85,B 0,C 180,E1 -7920,E2 -7920} C_VEL
LIN {X 0,Y 460.82,Z 376.582,A -85,B 0,C 180,E1 -7922.623,E2 -7922.623} C_VEL
LIN {X 0,Y 460.704,Z 376.599,A -85,B 0,C 180,E1 -7926.13,E2 -7926.13} C_VEL
LIN {X 0,Y 460.623,Z 376.587,A -85,B 0,C 180,E1 -7928.777,E2 -7928.777} C_VEL
LIN {X 0,Y 460.608,Z 376.61,A -85,B 0,C 180,E1 -7932.446,E2 -7932.446} C_VEL
LIN {X 0,Y 460.617,Z 376.607,A -85,B 0,C 180,E1 -7936.008,E2 -7936.008} C_VEL
LIN {X 0,Y 460.565,Z 376.6,A -85,B 0,C 180,E1 -7939.616,E2 -7939.616} C_VEL
LIN {X 0,Y 460.508,Z 376.622,A -85,B 0,C 180,E1 -7942.429,E2 -7942.429} C_VEL
LIN {X 0,Y 460.565,Z 376.608,A -85,B 0,C 180,E1 -7945.803,E2 -7945.803} C_VEL
LIN {X 0,Y 460.555,Z 376.611,A -85,B 0,C 180,E1 -7948.233,E2 -7948.233} C_VEL
LIN {X 0,Y 460.522,Z 376.617,A -85,B 0,C 180,E1 -7951.285,E2 -7951.285} C_VEL
LIN {X 0,Y 460.531,Z 376.614,A -85,B 0,C 180,E1 -7954.507,E2 -7954.507} C_VEL
LIN {X 0,Y 460.527,Z 376.619,A -85,B 0,C 180,E1 -7957.621,E2 -7957.621} C_VEL
LIN {X 0,Y 460.557,Z 376.613,A -85,B 0,C 180,E1 -7960.273,E2 -7960.273} C_VEL
LIN {X 0,Y 460.523,Z 376.617,A -85,B 0,C 180,E1 -7963.373,E2 -7963.373} C_VEL
LIN {X 0,Y 460.498,Z 376.621,A -85,B 0,C 180,E1 -7966.625,E2 -7966.625} C_VEL
LIN {X 0,Y 460.541,Z 376.605,A -85,B 0,C 180,E1 -7969.731,E2 -7969.731} C_VEL
LIN {X 0,Y 460.527,Z 376.617,A -85,B 0,C 180,E1 -7972.52,E2 -7972.52} C_VEL
LIN {X 0,Y 460.549,Z 376.617,A -85,B 0,C 180,E1 -7975.625,E2 -7975.625} C_VEL
LIN {X 0,Y 460.538,Z 376.619,A -85,B 0,C 180,E1 -7978.745,E2 -7978.745} C_VEL
LIN {X 0,Y 460.603,Z 376.733,A -85,B 0,C 180,E1 -7982.219,E2 -7982.219} C_VEL
LIN {X 0,Y 462.197,Z 385.104,A -85,B 0,C 180,E1 -7984.347,E2 -7984.347} C_VEL
LIN {X 0,Y 462.451,Z 390.071,A -85,B 0,C 180,E1 -7985.536,E2 -7985.536} C_VEL
LIN {X 0,Y 461.74,Z 404.571,A -85,B 0,C 180,E1 -7988.809,E2 -7988.809} C_VEL
LIN {X 0,Y 461.175,Z 417.963,A -85,B 0,C 180,E1 -7991.796,E2 -7991.796} C_VEL
LIN {X 0,Y 460.937,Z 421.898,A -85,B 0,C 180,E1 -7992.675,E2 -7992.675} C_VEL
LIN {X 0,Y 461.536,Z 425.487,A -85,B 0,C 180,E1 -7992.803,E2 -7992.803} C_VEL
LIN {X 0,Y 464.424,Z 442.274,A -85,B 0,C 180,E1 -7993.177,E2 -7993.177} C_VEL
LIN {X 0,Y 463.746,Z 526.858,A -85,B 0,C 180,E1 -7994.508,E2 -7994.508} C_VEL
LIN {X 0,Y 463.534,Z 536.772,A -85,B 0,C 180,E1 -7994.755,E2 -7994.755} C_VEL
LIN {X 0,Y 463.132,Z 546.757,A -85,B 0,C 180,E1 -7995.107,E2 -7995.107} C_VEL
LIN {X 0,Y 462.738,Z 557.115,A -85,B 0,C 180,E1 -7995.6,E2 -7995.6} C_VEL
LIN {X 0,Y 462.305,Z 566.262,A -85,B 0,C 180,E1 -7996.147,E2 -7996.147} C_VEL
LIN {X 0,Y 461.893,Z 575.267,A -85,B 0,C 180,E1 -7996.807,E2 -7996.807} C_VEL
LIN {X 0,Y 461.555,Z 583.486,A -85,B 0,C 180,E1 -7997.528,E2 -7997.528} C_VEL
LIN {X 0,Y 461.159,Z 591.423,A -85,B 0,C 180,E1 -7998.351,E2 -7998.351} C_VEL
LIN {X 0,Y 460.614,Z 600.219,A -85,B 0,C 180,E1 -7999.45,E2 -7999.45} C_VEL
LIN {X 0,Y 460.361,Z 606.211,A -85,B 0,C 180,E1 -8000.333,E2 -8000.333} C_VEL
LIN {X 0,Y 460.054,Z 612.522,A -85,B 0,C 180,E1 -8001.435,E2 -8001.435} C_VEL
LIN {X 0,Y 459.86,Z 617.795,A -85,B 0,C 180,E1 -8002.536,E2 -8002.536} C_VEL
LIN {X 0,Y 459.673,Z 622.886,A -85,B 0,C 180,E1 -8003.857,E2 -8003.857} C_VEL
LIN {X 0,Y 459.618,Z 626.848,A -85,B 0,C 180,E1 -8005.176,E2 -8005.176} C_VEL
LIN {X 0,Y 459.584,Z 629.778,A -85,B 0,C 180,E1 -8006.493,E2 -8006.493} C_VEL
LIN {X 0,Y 459.584,Z 631.276,A -85,B 0,C 180,E1 -8007.371,E2 -8007.371} C_VEL
LIN {X 0,Y 459.522,Z 632.793,A -85,B 0,C 180,E1 -8009.124,E2 -8009.124} C_VEL
LIN {X 0,Y 459.53,Z 633.072,A -85,B 0,C 180,E1 -8010,E2 -8010} C_VEL
LIN {X 0,Y 459.52,Z 632.199,A -85,B 0,C 180,E1 -8011.753,E2 -8011.753} C_VEL
LIN {X 0,Y 459.584,Z 631.275,A -85,B 0,C 180,E1 -8012.63,E2 -8012.63} C_VEL
LIN {X 0,Y 459.565,Z 627.933,A -85,B 0,C 180,E1 -8014.386,E2 -8014.386} C_VEL
LIN {X 0,Y 459.667,Z 624.312,A -85,B 0,C 180,E1 -8015.704,E2 -8015.704} C_VEL
LIN {X 0,Y 459.74,Z 621.373,A -85,B 0,C 180,E1 -8016.583,E2 -8016.583} C_VEL
LIN {X 0,Y 459.934,Z 615.797,A -85,B 0,C 180,E1 -8017.905,E2 -8017.905} C_VEL
LIN {X 0,Y 460.157,Z 610.143,A -85,B 0,C 180,E1 -8019.007,E2 -8019.007} C_VEL
LIN {X 0,Y 460.483,Z 603.338,A -85,B 0,C 180,E1 -8020.109,E2 -8020.109} C_VEL
LIN {X 0,Y 460.922,Z 595.119,A -85,B 0,C 180,E1 -8021.21,E2 -8021.21} C_VEL
LIN {X 0,Y 461.348,Z 587.29,A -85,B 0,C 180,E1 -8022.091,E2 -8022.091} C_VEL
LIN {X 0,Y 461.762,Z 578.566,A -85,B 0,C 180,E1 -8022.916,E2 -8022.916} C_VEL
LIN {X 0,Y 462.229,Z 569.438,A -85,B 0,C 180,E1 -8023.631,E2 -8023.631} C_VEL
LIN {X 0,Y 462.583,Z 561.044,A -85,B 0,C 180,E1 -8024.181,E2 -8024.181} C_VEL
LIN {X 0,Y 463.055,Z 550.535,A -85,B 0,C 180,E1 -8024.728,E2 -8024.728} C_VEL
LIN {X 0,Y 463.357,Z 540.198,A -85,B 0,C 180,E1 -8025.139,E2 -8025.139} C_VEL
LIN {X 0,Y 463.73,Z 529.477,A -85,B 0,C 180,E1 -8025.436,E2 -8025.436} C_VEL
LIN {X 0,Y 463.969,Z 505.391,A -85,B 0,C 180,E1 -8025.843,E2 -8025.843} C_VEL
LIN {X 0,Y 464.298,Z 441.6,A -85,B 0,C 180,E1 -8026.838,E2 -8026.838} C_VEL
LIN {X 0,Y 460.986,Z 422.34,A -85,B 0,C 180,E1 -8027.285,E2 -8027.285} C_VEL
LIN {X 0,Y 460.979,Z 421.199,A -85,B 0,C 180,E1 -8027.444,E2 -8027.444} C_VEL
LIN {X 0,Y 461.472,Z 409.891,A -85,B 0,C 180,E1 -8030.039,E2 -8030.039} C_VEL
LIN {X 0,Y 462.148,Z 396.417,A -85,B 0,C 180,E1 -8033.053,E2 -8033.053} C_VEL
LIN {X 0,Y 462.519,Z 388.059,A -85,B 0,C 180,E1 -8034.94,E2 -8034.94} C_VEL
LIN {X 0,Y 461.411,Z 380.879,A -85,B 0,C 180,E1 -8036.701,E2 -8036.701} C_VEL
LIN {X 0,Y 460.603,Z 376.718,A -85,B 0,C 180,E1 -8037.805,E2 -8037.805} C_VEL
LIN {X 0,Y 460.54,Z 376.619,A -85,B 0,C 180,E1 -8041.255,E2 -8041.255} C_VEL
LIN {X 0,Y 460.537,Z 376.617,A -85,B 0,C 180,E1 -8044.506,E2 -8044.506} C_VEL
LIN {X 0,Y 460.531,Z 376.618,A -85,B 0,C 180,E1 -8047.62,E2 -8047.62} C_VEL
LIN {X 0,Y 460.544,Z 376.605,A -85,B 0,C 180,E1 -8050.269,E2 -8050.269} C_VEL
LIN {X 0,Y 460.501,Z 376.62,A -85,B 0,C 180,E1 -8053.375,E2 -8053.375} C_VEL
LIN {X 0,Y 460.526,Z 376.617,A -85,B 0,C 180,E1 -8056.627,E2 -8056.627} C_VEL
LIN {X 0,Y 460.56,Z 376.613,A -85,B 0,C 180,E1 -8059.728,E2 -8059.728} C_VEL
LIN {X 0,Y 460.528,Z 376.617,A -85,B 0,C 180,E1 -8062.519,E2 -8062.519} C_VEL
LIN {X 0,Y 460.548,Z 376.611,A -85,B 0,C 180,E1 -8065.623,E2 -8065.623} C_VEL
LIN {X 0,Y 460.537,Z 376.615,A -85,B 0,C 180,E1 -8068.744,E2 -8068.744} C_VEL
LIN {X 0,Y 460.558,Z 376.611,A -85,B 0,C 180,E1 -8071.767,E2 -8071.767} C_VEL
LIN {X 0,Y 460.558,Z 376.606,A -85,B 0,C 180,E1 -8074.705,E2 -8074.705} C_VEL
LIN {X 0,Y 460.512,Z 376.622,A -85,B 0,C 180,E1 -8077.571,E2 -8077.571} C_VEL
LIN {X 0,Y 460.568,Z 376.599,A -85,B 0,C 180,E1 -8080.384,E2 -8080.384} C_VEL
LIN {X 0,Y 460.63,Z 376.605,A -85,B 0,C 180,E1 -8084.059,E2 -8084.059} C_VEL
LIN {X 0,Y 460.607,Z 376.608,A -85,B 0,C 180,E1 -8087.665,E2 -8087.665} C_VEL
LIN {X 0,Y 460.627,Z 376.585,A -85,B 0,C 180,E1 -8091.223,E2 -8091.223} C_VEL
LIN {X 0,Y 460.708,Z 376.599,A -85,B 0,C 180,E1 -8093.87,E2 -8093.87} C_VEL
LIN {X 0,Y 460.822,Z 376.582,A -85,B 0,C 180,E1 -8097.377,E2 -8097.377} C_VEL
LIN {X 0,Y 460.85,Z 376.561,A -85,B 0,C 180,E1 -8100,E2 -8100} C_VEL
LIN {X 0,Y 460.823,Z 376.573,A -85,B 0,C 180,E1 -8102.622,E2 -8102.622} C_VEL
LIN {X 0,Y 460.707,Z 376.594,A -85,B 0,C 180,E1 -8106.129,E2 -8106.129} C_VEL
LIN {X 0,Y 460.626,Z 376.595,A -85,B 0,C 180,E1 -8108.776,E2 -8108.776} C_VEL
LIN {X 0,Y 460.631,Z 376.599,A -85,B 0,C 180,E1 -8112.456,E2 -8112.456} C_VEL
LIN {X 0,Y 460.597,Z 376.607,A -85,B 0,C 180,E1 -8115.997,E2 -8115.997} C_VEL
LIN {X 0,Y 460.567,Z 376.6,A -85,B 0,C 180,E1 -8118.901,E2 -8118.901} C_VEL
LIN {X 0,Y 460.512,Z 376.618,A -85,B 0,C 180,E1 -8121.485,E2 -8121.485} C_VEL
LIN {X 0,Y 460.539,Z 376.614,A -85,B 0,C 180,E1 -8124.332,E2 -8124.332} C_VEL
LIN {X 0,Y 460.58,Z 376.603,A -85,B 0,C 180,E1 -8127.243,E2 -8127.243} C_VEL
LIN {X 0,Y 460.507,Z 376.619,A -85,B 0,C 180,E1 -8130.24,E2 -8130.24} C_VEL
LIN {X 0,Y 460.525,Z 376.616,A -85,B 0,C 180,E1 -8133.324,E2 -8133.324} C_VEL
LIN {X 0,Y 460.475,Z 376.621,A -85,B 0,C 180,E1 -8136.529,E2 -8136.529} C_VEL
LIN {X 0,Y 460.541,Z 376.617,A -85,B 0,C 180,E1 -8138.897,E2 -8138.897} C_VEL
LIN {X 0,Y 460.52,Z 376.616,A -85,B 0,C 180,E1 -8142.181,E2 -8142.181} C_VEL
LIN {X 0,Y 460.512,Z 376.614,A -85,B 0,C 180,E1 -8145.411,E2 -8145.411} C_VEL
LIN {X 0,Y 460.531,Z 376.594,A -85,B 0,C 180,E1 -8148.397,E2 -8148.397} C_VEL
LIN {X 0,Y 460.54,Z 376.619,A -85,B 0,C 180,E1 -8151.269,E2 -8151.269} C_VEL
LIN {X 0,Y 460.51,Z 376.612,A -85,B 0,C 180,E1 -8154.554,E2 -8154.554} C_VEL
LIN {X 0,Y 460.529,Z 376.619,A -85,B 0,C 180,E1 -8157.716,E2 -8157.716} C_VEL
LIN {X 0,Y 460.544,Z 376.607,A -85,B 0,C 180,E1 -8160.769,E2 -8160.769} C_VEL
LIN {X 0,Y 460.56,Z 376.616,A -85,B 0,C 180,E1 -8163.735,E2 -8163.735} C_VEL
LIN {X 0,Y 460.542,Z 376.618,A -85,B 0,C 180,E1 -8166.624,E2 -8166.624} C_VEL
LIN {X 0,Y 460.549,Z 376.619,A -85,B 0,C 180,E1 -8169.453,E2 -8169.453} C_VEL
LIN {X 0,Y 460.556,Z 376.615,A -85,B 0,C 180,E1 -8172.23,E2 -8172.23} C_VEL
LIN {X 0,Y 460.562,Z 376.618,A -85,B 0,C 180,E1 -8174.965,E2 -8174.965} C_VEL
LIN {X 0,Y 460.608,Z 376.611,A -85,B 0,C 180,E1 -8178.559,E2 -8178.559} C_VEL
LIN {X 0,Y 460.574,Z 376.615,A -85,B 0,C 180,E1 -8179.231,E2 -8179.231} C_VEL
LIN {X 0,Y 459.919,Z 376.7,A -85,B 0,C 180,E1 -8179.961,E2 -8179.961} C_VEL
LIN {X 0,Y 457.101,Z 377.054,A -85,B 0,C 180,E1 -8181.148,E2 -8181.148} C_VEL
LIN {X 0,Y 454.722,Z 377.349,A -85,B 0,C 180,E1 -8182.105,E2 -8182.105} C_VEL
LIN {X 0,Y 453.711,Z 377.472,A -85,B 0,C 180,E1 -8182.844,E2 -8182.844} C_VEL
LIN {X 0,Y 453.634,Z 377.48,A -85,B 0,C 180,E1 -8183.094,E2 -8183.094} C_VEL
LIN {X 0,Y 453.669,Z 377.477,A -85,B 0,C 180,E1 -8184.667,E2 -8184.667} C_VEL
LIN {X 0,Y 453.762,Z 377.465,A -85,B 0,C 180,E1 -8187.337,E2 -8187.337} C_VEL
LIN {X 0,Y 453.821,Z 377.456,A -85,B 0,C 180,E1 -8190,E2 -8190} C_VEL
LIN {X 0,Y 453.762,Z 377.465,A -85,B 0,C 180,E1 -8192.663,E2 -8192.663} C_VEL
LIN {X 0,Y 453.675,Z 377.474,A -85,B 0,C 180,E1 -8196.225,E2 -8196.225} C_VEL
LIN {X 0,Y 453.589,Z 377.487,A -85,B 0,C 180,E1 -8198.913,E2 -8198.913} C_VEL
LIN {X 0,Y 453.559,Z 377.49,A -85,B 0,C 180,E1 -8202.529,E2 -8202.529} C_VEL
LIN {X 0,Y 453.54,Z 377.49,A -85,B 0,C 180,E1 -8206.196,E2 -8206.196} C_VEL
LIN {X 0,Y 453.516,Z 377.496,A -85,B 0,C 180,E1 -8209.041,E2 -8209.041} C_VEL
LIN {X 0,Y 453.471,Z 377.498,A -85,B 0,C 180,E1 -8211.836,E2 -8211.836} C_VEL
LIN {X 0,Y 453.509,Z 377.497,A -85,B 0,C 180,E1 -8214.734,E2 -8214.734} C_VEL
LIN {X 0,Y 453.533,Z 377.488,A -85,B 0,C 180,E1 -8217.961,E2 -8217.961} C_VEL
LIN {X 0,Y 453.478,Z 377.495,A -85,B 0,C 180,E1 -8220.759,E2 -8220.759} C_VEL
LIN {X 0,Y 453.472,Z 377.487,A -85,B 0,C 180,E1 -8223.912,E2 -8223.912} C_VEL
LIN {X 0,Y 453.465,Z 377.499,A -85,B 0,C 180,E1 -8227.188,E2 -8227.188} C_VEL
LIN {X 0,Y 453.524,Z 377.485,A -85,B 0,C 180,E1 -8229.445,E2 -8229.445} C_VEL
LIN {X 0,Y 453.455,Z 377.481,A -85,B 0,C 180,E1 -8232.995,E2 -8232.995} C_VEL
LIN {X 0,Y 453.466,Z 377.495,A -85,B 0,C 180,E1 -8235.78,E2 -8235.78} C_VEL
LIN {X 0,Y 453.508,Z 377.484,A -85,B 0,C 180,E1 -8239.406,E2 -8239.406} C_VEL
LIN {X 0,Y 453.467,Z 377.499,A -85,B 0,C 180,E1 -8242.223,E2 -8242.223} C_VEL
LIN {X 0,Y 453.482,Z 377.485,A -85,B 0,C 180,E1 -8245.222,E2 -8245.222} C_VEL
LIN {X 0,Y 453.477,Z 377.5,A -85,B 0,C 180,E1 -8248.471,E2 -8248.471} C_VEL
LIN {X 0,Y 453.508,Z 377.483,A -85,B 0,C 180,E1 -8251.289,E2 -8251.289} C_VEL
LIN {X 0,Y 453.518,Z 377.485,A -85,B 0,C 180,E1 -8254.285,E2 -8254.285} C_VEL
LIN {X 0,Y 453.473,Z 377.495,A -85,B 0,C 180,E1 -8257.204,E2 -8257.204} C_VEL
LIN {X 0,Y 453.498,Z 377.485,A -85,B 0,C 180,E1 -8260.066,E2 -8260.066} C_VEL
LIN {X 0,Y 453.5,Z 377.491,A -85,B 0,C 180,E1 -8262.876,E2 -8262.876} C_VEL
LIN {X 0,Y 453.506,Z 377.491,A -85,B 0,C 180,E1 -8265.644,E2 -8265.644} C_VEL
LIN {X 0,Y 453.571,Z 377.476,A -85,B 0,C 180,E1 -8268.38,E2 -8268.38} C_VEL
LIN {X 0,Y 453.645,Z 377.466,A -85,B 0,C 180,E1 -8271.986,E2 -8271.986} C_VEL
LIN {X 0,Y 453.666,Z 377.474,A -85,B 0,C 180,E1 -8274.667,E2 -8274.667} C_VEL
LIN {X 0,Y 453.76,Z 377.453,A -85,B 0,C 180,E1 -8277.337,E2 -8277.337} C_VEL
LIN {X 0,Y 453.817,Z 377.436,A -85,B 0,C 180,E1 -8280.001,E2 -8280.001} C_VEL
LIN {X 0,Y 453.76,Z 377.461,A -85,B 0,C 180,E1 -8282.664,E2 -8282.664} C_VEL
LIN {X 0,Y 453.672,Z 377.473,A -85,B 0,C 180,E1 -8286.226,E2 -8286.226} C_VEL
LIN {X 0,Y 453.587,Z 377.462,A -85,B 0,C 180,E1 -8288.914,E2 -8288.914} C_VEL
LIN {X 0,Y 453.558,Z 377.487,A -85,B 0,C 180,E1 -8292.529,E2 -8292.529} C_VEL
LIN {X 0,Y 453.551,Z 377.484,A -85,B 0,C 180,E1 -8296.196,E2 -8296.196} C_VEL
LIN {X 0,Y 453.516,Z 377.476,A -85,B 0,C 180,E1 -8299.041,E2 -8299.041} C_VEL
LIN {X 0,Y 453.472,Z 377.495,A -85,B 0,C 180,E1 -8301.837,E2 -8301.837} C_VEL
LIN {X 0,Y 453.51,Z 377.485,A -85,B 0,C 180,E1 -8304.735,E2 -8304.735} C_VEL
LIN {X 0,Y 453.535,Z 377.481,A -85,B 0,C 180,E1 -8307.962,E2 -8307.962} C_VEL
LIN {X 0,Y 453.48,Z 377.495,A -85,B 0,C 180,E1 -8310.76,E2 -8310.76} C_VEL
LIN {X 0,Y 453.475,Z 377.489,A -85,B 0,C 180,E1 -8313.913,E2 -8313.913} C_VEL
LIN {X 0,Y 453.469,Z 377.496,A -85,B 0,C 180,E1 -8317.189,E2 -8317.189} C_VEL
LIN {X 0,Y 453.526,Z 377.485,A -85,B 0,C 180,E1 -8319.446,E2 -8319.446} C_VEL
LIN {X 0,Y 453.49,Z 377.492,A -85,B 0,C 180,E1 -8322.992,E2 -8322.992} C_VEL
LIN {X 0,Y 453.465,Z 377.5,A -85,B 0,C 180,E1 -8325.78,E2 -8325.78} C_VEL
LIN {X 0,Y 453.478,Z 377.488,A -85,B 0,C 180,E1 -8328.21,E2 -8328.21} C_VEL
LIN {X 0,Y 453.509,Z 377.49,A -85,B 0,C 180,E1 -8330.792,E2 -8330.792} C_VEL
LIN {X 0,Y 453.457,Z 377.494,A -85,B 0,C 180,E1 -8333.918,E2 -8333.918} C_VEL
LIN {X 0,Y 453.483,Z 377.492,A -85,B 0,C 180,E1 -8337.152,E2 -8337.152} C_VEL
LIN {X 0,Y 453.515,Z 377.492,A -85,B 0,C 180,E1 -8340.272,E2 -8340.272} C_VEL
LIN {X 0,Y 453.579,Z 377.685,A -85,B 0,C 180,E1 -8342.03,E2 -8342.03} C_VEL
LIN {X 0,Y 455.452,Z 387.919,A -85,B 0,C 180,E1 -8344.647,E2 -8344.647} C_VEL
LIN {X 0,Y 455.291,Z 395.08,A -85,B 0,C 180,E1 -8346.338,E2 -8346.338} C_VEL
LIN {X 0,Y 454.532,Z 409.57,A -85,B 0,C 180,E1 -8349.642,E2 -8349.642} C_VEL
LIN {X 0,Y 453.959,Z 421.706,A -85,B 0,C 180,E1 -8352.4,E2 -8352.4} C_VEL
LIN {X 0,Y 454.476,Z 424.885,A -85,B 0,C 180,E1 -8352.521,E2 -8352.521} C_VEL
LIN {X 0,Y 457.609,Z 443.492,A -85,B 0,C 180,E1 -8352.942,E2 -8352.942} C_VEL
LIN {X 0,Y 456.918,Z 526.663,A -85,B 0,C 180,E1 -8354.271,E2 -8354.271} C_VEL
LIN {X 0,Y 456.706,Z 536.578,A -85,B 0,C 180,E1 -8354.521,E2 -8354.521} C_VEL
LIN {X 0,Y 456.276,Z 546.562,A -85,B 0,C 180,E1 -8354.878,E2 -8354.878} C_VEL
LIN {X 0,Y 455.867,Z 556.92,A -85,B 0,C 180,E1 -8355.378,E2 -8355.378} C_VEL
LIN {X 0,Y 455.406,Z 566.067,A -85,B 0,C 180,E1 -8355.933,E2 -8355.933} C_VEL
LIN {X 0,Y 454.974,Z 575.072,A -85,B 0,C 180,E1 -8356.603,E2 -8356.603} C_VEL
LIN {X 0,Y 454.588,Z 583.474,A -85,B 0,C 180,E1 -8357.353,E2 -8357.353} C_VEL
LIN {X 0,Y 454.15,Z 591.226,A -85,B 0,C 180,E1 -8358.168,E2 -8358.168} C_VEL
LIN {X 0,Y 453.608,Z 600.023,A -85,B 0,C 180,E1 -8359.285,E2 -8359.285} C_VEL
LIN {X 0,Y 453.33,Z 606.015,A -85,B 0,C 180,E1 -8360.182,E2 -8360.182} C_VEL
LIN {X 0,Y 453.013,Z 612.326,A -85,B 0,C 180,E1 -8361.3,E2 -8361.3} C_VEL
LIN {X 0,Y 452.808,Z 617.6,A -85,B 0,C 180,E1 -8362.419,E2 -8362.419} C_VEL
LIN {X 0,Y 452.605,Z 622.691,A -85,B 0,C 180,E1 -8363.76,E2 -8363.76} C_VEL
LIN {X 0,Y 452.547,Z 626.653,A -85,B 0,C 180,E1 -8365.1,E2 -8365.1} C_VEL
LIN {X 0,Y 452.48,Z 629.583,A -85,B 0,C 180,E1 -8366.438,E2 -8366.438} C_VEL
LIN {X 0,Y 452.508,Z 631.081,A -85,B 0,C 180,E1 -8367.33,E2 -8367.33} C_VEL
LIN {X 0,Y 452.428,Z 632.598,A -85,B 0,C 180,E1 -8369.11,E2 -8369.11} C_VEL
LIN {X 0,Y 452.434,Z 632.877,A -85,B 0,C 180,E1 -8370,E2 -8370} C_VEL
LIN {X 0,Y 452.437,Z 632.004,A -85,B 0,C 180,E1 -8371.781,E2 -8371.781} C_VEL
LIN {X 0,Y 452.508,Z 631.08,A -85,B 0,C 180,E1 -8372.671,E2 -8372.671} C_VEL
LIN {X 0,Y 452.487,Z 627.738,A -85,B 0,C 180,E1 -8374.454,E2 -8374.454} C_VEL
LIN {X 0,Y 452.569,Z 625.528,A -85,B 0,C 180,E1 -8375.346,E2 -8375.346} C_VEL
LIN {X 0,Y 452.651,Z 621.349,A -85,B 0,C 180,E1 -8376.643,E2 -8376.643} C_VEL
LIN {X 0,Y 452.869,Z 615.601,A -85,B 0,C 180,E1 -8378.029,E2 -8378.029} C_VEL
LIN {X 0,Y 453.111,Z 609.947,A -85,B 0,C 180,E1 -8379.148,E2 -8379.148} C_VEL
LIN {X 0,Y 453.449,Z 603.141,A -85,B 0,C 180,E1 -8380.267,E2 -8380.267} C_VEL
LIN {X 0,Y 453.941,Z 594.924,A -85,B 0,C 180,E1 -8381.385,E2 -8381.385} C_VEL
LIN {X 0,Y 454.385,Z 587.094,A -85,B 0,C 180,E1 -8382.279,E2 -8382.279} C_VEL
LIN {X 0,Y 454.829,Z 578.37,A -85,B 0,C 180,E1 -8383.116,E2 -8383.116} C_VEL
LIN {X 0,Y 455.308,Z 569.242,A -85,B 0,C 180,E1 -8383.843,E2 -8383.843} C_VEL
LIN {X 0,Y 455.685,Z 560.848,A -85,B 0,C 180,E1 -8384.4,E2 -8384.4} C_VEL
LIN {X 0,Y 456.196,Z 550.34,A -85,B 0,C 180,E1 -8384.954,E2 -8384.954} C_VEL
LIN {X 0,Y 456.498,Z 540.003,A -85,B 0,C 180,E1 -8385.372,E2 -8385.372} C_VEL
LIN {X 0,Y 456.904,Z 529.282,A -85,B 0,C 180,E1 -8385.673,E2 -8385.673} C_VEL
LIN {X 0,Y 457.15,Z 505.274,A -85,B 0,C 180,E1 -8386.084,E2 -8386.084} C_VEL
LIN {X 0,Y 457.51,Z 442.494,A -85,B 0,C 180,E1 -8387.078,E2 -8387.078} C_VEL
LIN {X 0,Y 454.014,Z 422.136,A -85,B 0,C 180,E1 -8387.559,E2 -8387.559} C_VEL
LIN {X 0,Y 454.003,Z 420.648,A -85,B 0,C 180,E1 -8387.808,E2 -8387.808} C_VEL
LIN {X 0,Y 454.631,Z 408.701,A -85,B 0,C 180,E1 -8390.59,E2 -8390.59} C_VEL
LIN {X 0,Y 455.398,Z 393.518,A -85,B 0,C 180,E1 -8394.051,E2 -8394.051} C_VEL
LIN {X 0,Y 455.455,Z 387.917,A -85,B 0,C 180,E1 -8395.353,E2 -8395.353} C_VEL
LIN {X 0,Y 453.572,Z 377.593,A -85,B 0,C 180,E1 -8398.026,E2 -8398.026} C_VEL
LIN {X 0,Y 453.486,Z 377.499,A -85,B 0,C 180,E1 -8400.759,E2 -8400.759} C_VEL
LIN {X 0,Y 453.481,Z 377.499,A -85,B 0,C 180,E1 -8403.912,E2 -8403.912} C_VEL
LIN {X 0,Y 453.473,Z 377.494,A -85,B 0,C 180,E1 -8407.188,E2 -8407.188} C_VEL
LIN {X 0,Y 453.507,Z 377.492,A -85,B 0,C 180,E1 -8409.448,E2 -8409.448} C_VEL
LIN {X 0,Y 453.464,Z 377.495,A -85,B 0,C 180,E1 -8412.994,E2 -8412.994} C_VEL
LIN {X 0,Y 453.478,Z 377.495,A -85,B 0,C 180,E1 -8415.78,E2 -8415.78} C_VEL
LIN {X 0,Y 453.498,Z 377.495,A -85,B 0,C 180,E1 -8418.211,E2 -8418.211} C_VEL
LIN {X 0,Y 453.527,Z 377.484,A -85,B 0,C 180,E1 -8420.788,E2 -8420.788} C_VEL
LIN {X 0,Y 453.457,Z 377.5,A -85,B 0,C 180,E1 -8423.917,E2 -8423.917} C_VEL
LIN {X 0,Y 453.483,Z 377.487,A -85,B 0,C 180,E1 -8427.151,E2 -8427.151} C_VEL
LIN {X 0,Y 453.514,Z 377.491,A -85,B 0,C 180,E1 -8430.271,E2 -8430.271} C_VEL
LIN {X 0,Y 453.509,Z 377.48,A -85,B 0,C 180,E1 -8433.294,E2 -8433.294} C_VEL
LIN {X 0,Y 453.503,Z 377.493,A -85,B 0,C 180,E1 -8436.238,E2 -8436.238} C_VEL
LIN {X 0,Y 453.482,Z 377.491,A -85,B 0,C 180,E1 -8439.117,E2 -8439.117} C_VEL
LIN {X 0,Y 453.51,Z 377.48,A -85,B 0,C 180,E1 -8441.944,E2 -8441.944} C_VEL
LIN {X 0,Y 453.548,Z 377.483,A -85,B 0,C 180,E1 -8444.726,E2 -8444.726} C_VEL
